REGION Network 73: SN51_N0063
   RUNG wire#powerrail
      Contact( "AlwaysTRUE" )
      Contact( "ZAUX".SN51_N0063 )
      Coil( "00_Commissioning"."n0063-lv006-el001-k30001_SN51" )
   END_RUNG
   // the same network as SCL:
   "00_Commissioning"."n0063-lv006-el001-k30001_SN51" := "AlwaysTRUE" AND "ZAUX".SN51_N0063;
END_REGION

REGION Network 74: SN51_N0066
   RUNG wire#powerrail
      Contact( "AlwaysTRUE" )
      Contact( "ZAUX".SN51_N0066 )
      Coil( "00_Commissioning"."n0066-uc21-el001-k30001_SN51" )
   END_RUNG
   // the same network as SCL:
   "00_Commissioning"."n0066-uc21-el001-k30001_SN51" := "AlwaysTRUE" AND "ZAUX".SN51_N0066;
END_REGION

REGION Network 75: SN51_N0067
   RUNG wire#powerrail
      Contact( "AlwaysTRUE" )
      Contact( "ZAUX".SN51_N0067 )
      Coil( "00_Commissioning"."n0067-uc214-xn10_SN51" )
   END_RUNG
   // the same network as SCL:
   "00_Commissioning"."n0067-uc214-xn10_SN51" := "AlwaysTRUE" AND "ZAUX".SN51_N0067;
END_REGION

REGION Network 76: SN51_N0070
   RUNG wire#powerrail
      Contact( "AlwaysTRUE" )
      Contact( "ZAUX".SN51_N0070 )
      Coil( "00_Commissioning"."n0070-uf31-el001-k30001_SN51" )
   END_RUNG
   // the same network as SCL:
   "00_Commissioning"."n0070-uf31-el001-k30001_SN51" := "AlwaysTRUE" AND "ZAUX".SN51_N0070;
END_REGION

REGION Network 77: SN51_N0071
   RUNG wire#powerrail
      Contact( "AlwaysTRUE" )
      Contact( "ZAUX".SN51_N0071 )
      Coil( "00_Commissioning"."n0070-uf31-el001-k30001_SN51" )
   END_RUNG
   // the same network as SCL:
   "00_Commissioning"."n0070-uf31-el001-k30001_SN51" := "AlwaysTRUE" AND "ZAUX".SN51_N0071;
END_REGION

REGION Network 78: SN51_N0072
   RUNG wire#powerrail
      Contact( "AlwaysTRUE" )
      Contact( "ZAUX".SN51_N0072 )
      Coil( "00_Commissioning"."n0072-uf51-el001-k30001_SN51" )
   END_RUNG
   // the same network as SCL:
   "00_Commissioning"."n0072-uf51-el001-k30001_SN51" := "AlwaysTRUE" AND "ZAUX".SN51_N0072;
END_REGION

REGION Network 79: SN51_N0080
   RUNG wire#powerrail
      Contact( "AlwaysTRUE" )
      Contact( "ZAUX".SN51_N0080 )
      Coil( "00_Commissioning"."n0080-uf511-xn10_SN51" )
   END_RUNG
   // the same network as SCL:
   "00_Commissioning"."n0080-uf511-xn10_SN51" := "AlwaysTRUE" AND "ZAUX".SN51_N0080;
END_REGION

REGION Network 80: SN51_N0073
   RUNG wire#powerrail
      Contact( "AlwaysTRUE" )
      Contact( "ZAUX".SN51_N0073 )
      Coil( "00_Commissioning"."n0073-ifg31-el001-k30001_SN51" )
   END_RUNG
   // the same network as SCL:
   "00_Commissioning"."n0073-ifg31-el001-k30001_SN51" := "AlwaysTRUE" AND "ZAUX".SN51_N0073;
END_REGION

REGION Network 81: SN51_N0074
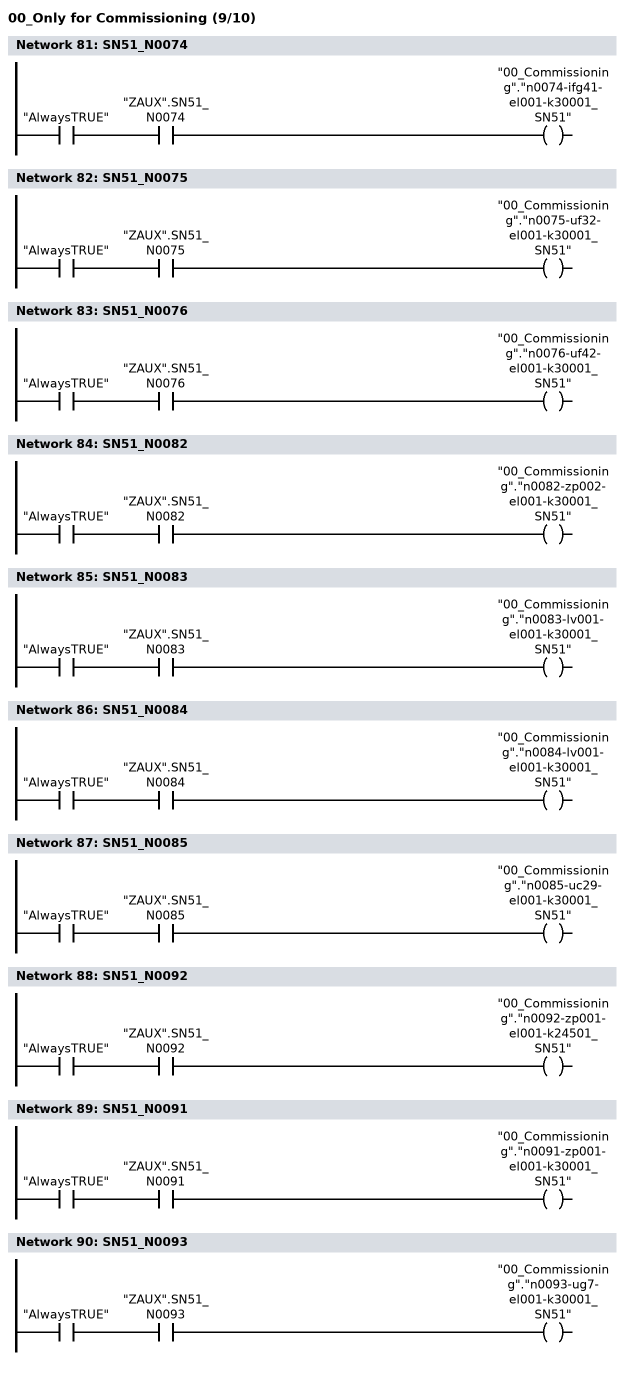
   RUNG wire#powerrail
      Contact( "AlwaysTRUE" )
      Contact( "ZAUX".SN51_N0074 )
      Coil( "00_Commissioning"."n0074-ifg41-el001-k30001_SN51" )
   END_RUNG
   // the same network as SCL:
   "00_Commissioning"."n0074-ifg41-el001-k30001_SN51" := "AlwaysTRUE" AND "ZAUX".SN51_N0074;
END_REGION

REGION Network 82: SN51_N0075
   RUNG wire#powerrail
      Contact( "AlwaysTRUE" )
      Contact( "ZAUX".SN51_N0075 )
      Coil( "00_Commissioning"."n0075-uf32-el001-k30001_SN51" )
   END_RUNG
   // the same network as SCL:
   "00_Commissioning"."n0075-uf32-el001-k30001_SN51" := "AlwaysTRUE" AND "ZAUX".SN51_N0075;
END_REGION

REGION Network 83: SN51_N0076
   RUNG wire#powerrail
      Contact( "AlwaysTRUE" )
      Contact( "ZAUX".SN51_N0076 )
      Coil( "00_Commissioning"."n0076-uf42-el001-k30001_SN51" )
   END_RUNG
   // the same network as SCL:
   "00_Commissioning"."n0076-uf42-el001-k30001_SN51" := "AlwaysTRUE" AND "ZAUX".SN51_N0076;
END_REGION

REGION Network 84: SN51_N0082
   RUNG wire#powerrail
      Contact( "AlwaysTRUE" )
      Contact( "ZAUX".SN51_N0082 )
      Coil( "00_Commissioning"."n0082-zp002-el001-k30001_SN51" )
   END_RUNG
   // the same network as SCL:
   "00_Commissioning"."n0082-zp002-el001-k30001_SN51" := "AlwaysTRUE" AND "ZAUX".SN51_N0082;
END_REGION

REGION Network 85: SN51_N0083
   RUNG wire#powerrail
      Contact( "AlwaysTRUE" )
      Contact( "ZAUX".SN51_N0083 )
      Coil( "00_Commissioning"."n0083-lv001-el001-k30001_SN51" )
   END_RUNG
   // the same network as SCL:
   "00_Commissioning"."n0083-lv001-el001-k30001_SN51" := "AlwaysTRUE" AND "ZAUX".SN51_N0083;
END_REGION

REGION Network 86: SN51_N0084
   RUNG wire#powerrail
      Contact( "AlwaysTRUE" )
      Contact( "ZAUX".SN51_N0084 )
      Coil( "00_Commissioning"."n0084-lv001-el001-k30001_SN51" )
   END_RUNG
   // the same network as SCL:
   "00_Commissioning"."n0084-lv001-el001-k30001_SN51" := "AlwaysTRUE" AND "ZAUX".SN51_N0084;
END_REGION

REGION Network 87: SN51_N0085
   RUNG wire#powerrail
      Contact( "AlwaysTRUE" )
      Contact( "ZAUX".SN51_N0085 )
      Coil( "00_Commissioning"."n0085-uc29-el001-k30001_SN51" )
   END_RUNG
   // the same network as SCL:
   "00_Commissioning"."n0085-uc29-el001-k30001_SN51" := "AlwaysTRUE" AND "ZAUX".SN51_N0085;
END_REGION

REGION Network 88: SN51_N0092
   RUNG wire#powerrail
      Contact( "AlwaysTRUE" )
      Contact( "ZAUX".SN51_N0092 )
      Coil( "00_Commissioning"."n0092-zp001-el001-k24501_SN51" )
   END_RUNG
   // the same network as SCL:
   "00_Commissioning"."n0092-zp001-el001-k24501_SN51" := "AlwaysTRUE" AND "ZAUX".SN51_N0092;
END_REGION

REGION Network 89: SN51_N0091
   RUNG wire#powerrail
      Contact( "AlwaysTRUE" )
      Contact( "ZAUX".SN51_N0091 )
      Coil( "00_Commissioning"."n0091-zp001-el001-k30001_SN51" )
   END_RUNG
   // the same network as SCL:
   "00_Commissioning"."n0091-zp001-el001-k30001_SN51" := "AlwaysTRUE" AND "ZAUX".SN51_N0091;
END_REGION

REGION Network 90: SN51_N0093
   RUNG wire#powerrail
      Contact( "AlwaysTRUE" )
      Contact( "ZAUX".SN51_N0093 )
      Coil( "00_Commissioning"."n0093-ug7-el001-k30001_SN51" )
   END_RUNG
   // the same network as SCL:
   "00_Commissioning"."n0093-ug7-el001-k30001_SN51" := "AlwaysTRUE" AND "ZAUX".SN51_N0093;
END_REGION

REGION Network 91: SN51_N0094
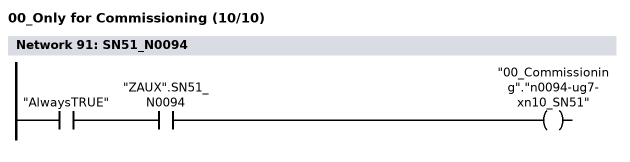
   RUNG wire#powerrail
      Contact( "AlwaysTRUE" )
      Contact( "ZAUX".SN51_N0094 )
      Coil( "00_Commissioning"."n0094-ug7-xn10_SN51" )
   END_RUNG
   // the same network as SCL:
   "00_Commissioning"."n0094-ug7-xn10_SN51" := "AlwaysTRUE" AND "ZAUX".SN51_N0094;
END_REGION
END_FUNCTION

FUNCTION "01_Settings" : Void   // FC2, F_FBD
{ S7_Optimized_Access := 'TRUE' }
VERSION : 0.1
BEGIN

REGION Network 1: To be used in case of overall settings
   // for example in case of Tristate diagnostic
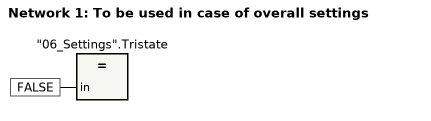
   "06_Settings".Tristate := FALSE;
END_REGION
END_FUNCTION

FUNCTION "02_EM Push Button" : Void   // FC3, F_LAD
TITLE = Mirror PB
{ S7_Optimized_Access := 'TRUE' }
VERSION : 0.1
BEGIN

REGION Network 1: 50.005 | n0005-zp001-el001-k40001_SN50 [1]
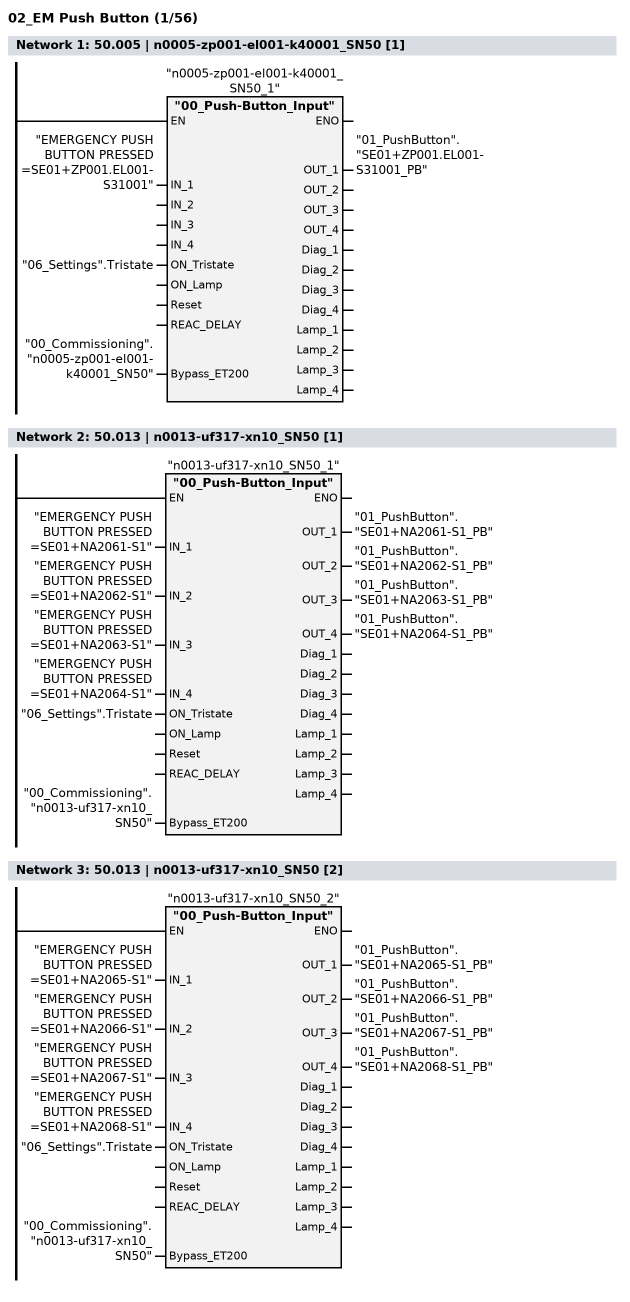
   RUNG wire#powerrail
      "n0005-zp001-el001-k40001_SN50_1"(IN_1 := "EMERGENCY PUSH BUTTON PRESSED =SE01+ZP001.EL001-S31001", IN_2 :=, IN_3 :=, IN_4 :=, ON_Tristate := "06_Settings".Tristate, ON_Lamp :=, Reset :=, REAC_DELAY :=, Bypass_ET200 := "00_Commissioning"."n0005-zp001-el001-k40001_SN50", OUT_1 => "01_PushButton"."SE01+ZP001.EL001-S31001_PB", OUT_2 =>, OUT_3 =>, OUT_4 =>, Diag_1 =>, Diag_2 =>, Diag_3 =>, Diag_4 =>, Lamp_1 =>, Lamp_2 =>, Lamp_3 =>, Lamp_4 =>)
   END_RUNG
   // the same network as SCL:
   "n0005-zp001-el001-k40001_SN50_1"(IN_1 := "EMERGENCY PUSH BUTTON PRESSED =SE01+ZP001.EL001-S31001",   // "00_Push-Button_Input"
                           ON_Tristate := "06_Settings".Tristate,
                           Bypass_ET200 := "00_Commissioning"."n0005-zp001-el001-k40001_SN50",
                           OUT_1 => "01_PushButton"."SE01+ZP001.EL001-S31001_PB");
END_REGION

REGION Network 2: 50.013 | n0013-uf317-xn10_SN50 [1]
   RUNG wire#powerrail
      "n0013-uf317-xn10_SN50_1"(IN_1 := "EMERGENCY PUSH BUTTON PRESSED =SE01+NA2061-S1", IN_2 := "EMERGENCY PUSH BUTTON PRESSED =SE01+NA2062-S1", IN_3 := "EMERGENCY PUSH BUTTON PRESSED =SE01+NA2063-S1", IN_4 := "EMERGENCY PUSH BUTTON PRESSED =SE01+NA2064-S1", ON_Tristate := "06_Settings".Tristate, ON_Lamp :=, Reset :=, REAC_DELAY :=, Bypass_ET200 := "00_Commissioning"."n0013-uf317-xn10_SN50", OUT_1 => "01_PushButton"."SE01+NA2061-S1_PB", OUT_2 => "01_PushButton"."SE01+NA2062-S1_PB", OUT_3 => "01_PushButton"."SE01+NA2063-S1_PB", OUT_4 => "01_PushButton"."SE01+NA2064-S1_PB", Diag_1 =>, Diag_2 =>, Diag_3 =>, Diag_4 =>, Lamp_1 =>, Lamp_2 =>, Lamp_3 =>, Lamp_4 =>)
   END_RUNG
   // the same network as SCL:
   "n0013-uf317-xn10_SN50_1"(IN_1 := "EMERGENCY PUSH BUTTON PRESSED =SE01+NA2061-S1",   // "00_Push-Button_Input"
                           IN_2 := "EMERGENCY PUSH BUTTON PRESSED =SE01+NA2062-S1",
                           IN_3 := "EMERGENCY PUSH BUTTON PRESSED =SE01+NA2063-S1",
                           IN_4 := "EMERGENCY PUSH BUTTON PRESSED =SE01+NA2064-S1",
                           ON_Tristate := "06_Settings".Tristate,
                           Bypass_ET200 := "00_Commissioning"."n0013-uf317-xn10_SN50",
                           OUT_1 => "01_PushButton"."SE01+NA2061-S1_PB",
                           OUT_2 => "01_PushButton"."SE01+NA2062-S1_PB",
                           OUT_3 => "01_PushButton"."SE01+NA2063-S1_PB",
                           OUT_4 => "01_PushButton"."SE01+NA2064-S1_PB");
END_REGION

REGION Network 3: 50.013 | n0013-uf317-xn10_SN50 [2]
   RUNG wire#powerrail
      "n0013-uf317-xn10_SN50_2"(IN_1 := "EMERGENCY PUSH BUTTON PRESSED =SE01+NA2065-S1", IN_2 := "EMERGENCY PUSH BUTTON PRESSED =SE01+NA2066-S1", IN_3 := "EMERGENCY PUSH BUTTON PRESSED =SE01+NA2067-S1", IN_4 := "EMERGENCY PUSH BUTTON PRESSED =SE01+NA2068-S1", ON_Tristate := "06_Settings".Tristate, ON_Lamp :=, Reset :=, REAC_DELAY :=, Bypass_ET200 := "00_Commissioning"."n0013-uf317-xn10_SN50", OUT_1 => "01_PushButton"."SE01+NA2065-S1_PB", OUT_2 => "01_PushButton"."SE01+NA2066-S1_PB", OUT_3 => "01_PushButton"."SE01+NA2067-S1_PB", OUT_4 => "01_PushButton"."SE01+NA2068-S1_PB", Diag_1 =>, Diag_2 =>, Diag_3 =>, Diag_4 =>, Lamp_1 =>, Lamp_2 =>, Lamp_3 =>, Lamp_4 =>)
   END_RUNG
   // the same network as SCL:
   "n0013-uf317-xn10_SN50_2"(IN_1 := "EMERGENCY PUSH BUTTON PRESSED =SE01+NA2065-S1",   // "00_Push-Button_Input"
                           IN_2 := "EMERGENCY PUSH BUTTON PRESSED =SE01+NA2066-S1",
                           IN_3 := "EMERGENCY PUSH BUTTON PRESSED =SE01+NA2067-S1",
                           IN_4 := "EMERGENCY PUSH BUTTON PRESSED =SE01+NA2068-S1",
                           ON_Tristate := "06_Settings".Tristate,
                           Bypass_ET200 := "00_Commissioning"."n0013-uf317-xn10_SN50",
                           OUT_1 => "01_PushButton"."SE01+NA2065-S1_PB",
                           OUT_2 => "01_PushButton"."SE01+NA2066-S1_PB",
                           OUT_3 => "01_PushButton"."SE01+NA2067-S1_PB",
                           OUT_4 => "01_PushButton"."SE01+NA2068-S1_PB");
END_REGION

REGION Network 4: 50.015 | n0015-uc16-el001-k30001_SN50 [1]
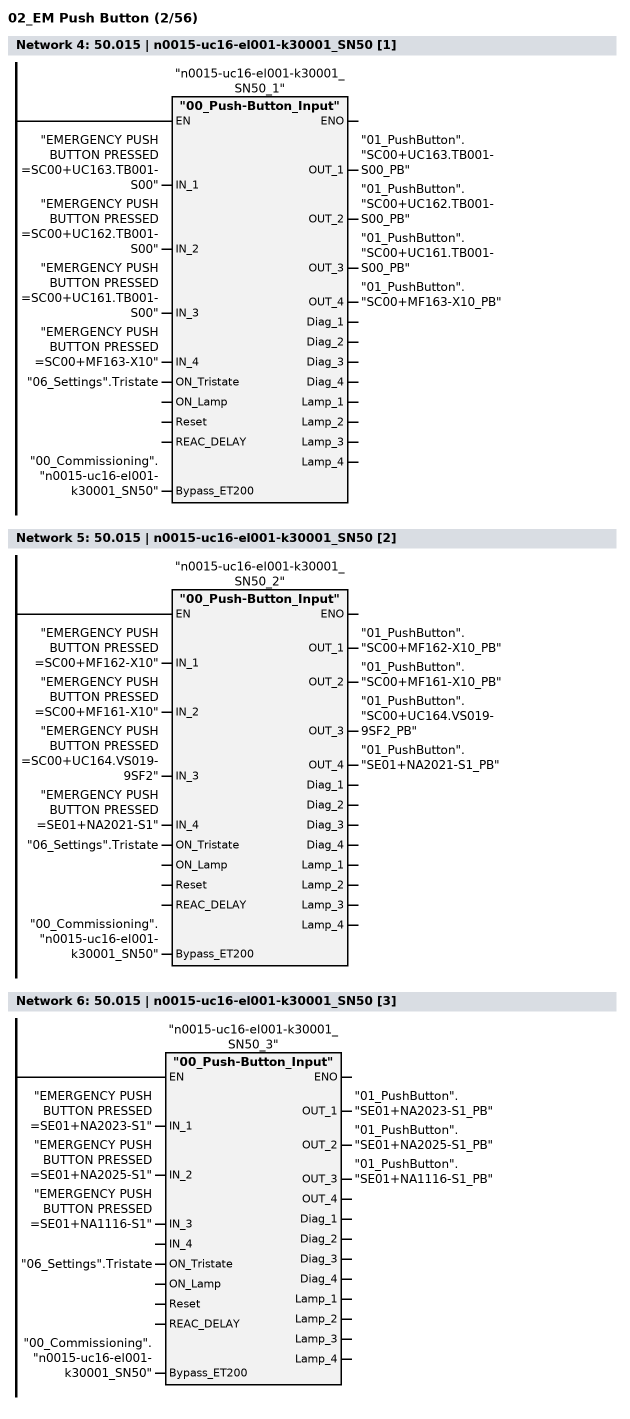
   RUNG wire#powerrail
      "n0015-uc16-el001-k30001_SN50_1"(IN_1 := "EMERGENCY PUSH BUTTON PRESSED =SC00+UC163.TB001-S00", IN_2 := "EMERGENCY PUSH BUTTON PRESSED =SC00+UC162.TB001-S00", IN_3 := "EMERGENCY PUSH BUTTON PRESSED =SC00+UC161.TB001-S00", IN_4 := "EMERGENCY PUSH BUTTON PRESSED =SC00+MF163-X10", ON_Tristate := "06_Settings".Tristate, ON_Lamp :=, Reset :=, REAC_DELAY :=, Bypass_ET200 := "00_Commissioning"."n0015-uc16-el001-k30001_SN50", OUT_1 => "01_PushButton"."SC00+UC163.TB001-S00_PB", OUT_2 => "01_PushButton"."SC00+UC162.TB001-S00_PB", OUT_3 => "01_PushButton"."SC00+UC161.TB001-S00_PB", OUT_4 => "01_PushButton"."SC00+MF163-X10_PB", Diag_1 =>, Diag_2 =>, Diag_3 =>, Diag_4 =>, Lamp_1 =>, Lamp_2 =>, Lamp_3 =>, Lamp_4 =>)
   END_RUNG
   // the same network as SCL:
   "n0015-uc16-el001-k30001_SN50_1"(IN_1 := "EMERGENCY PUSH BUTTON PRESSED =SC00+UC163.TB001-S00",   // "00_Push-Button_Input"
                           IN_2 := "EMERGENCY PUSH BUTTON PRESSED =SC00+UC162.TB001-S00",
                           IN_3 := "EMERGENCY PUSH BUTTON PRESSED =SC00+UC161.TB001-S00",
                           IN_4 := "EMERGENCY PUSH BUTTON PRESSED =SC00+MF163-X10",
                           ON_Tristate := "06_Settings".Tristate,
                           Bypass_ET200 := "00_Commissioning"."n0015-uc16-el001-k30001_SN50",
                           OUT_1 => "01_PushButton"."SC00+UC163.TB001-S00_PB",
                           OUT_2 => "01_PushButton"."SC00+UC162.TB001-S00_PB",
                           OUT_3 => "01_PushButton"."SC00+UC161.TB001-S00_PB",
                           OUT_4 => "01_PushButton"."SC00+MF163-X10_PB");
END_REGION

REGION Network 5: 50.015 | n0015-uc16-el001-k30001_SN50 [2]
   RUNG wire#powerrail
      "n0015-uc16-el001-k30001_SN50_2"(IN_1 := "EMERGENCY PUSH BUTTON PRESSED =SC00+MF162-X10", IN_2 := "EMERGENCY PUSH BUTTON PRESSED =SC00+MF161-X10", IN_3 := "EMERGENCY PUSH BUTTON PRESSED =SC00+UC164.VS019-9SF2", IN_4 := "EMERGENCY PUSH BUTTON PRESSED =SE01+NA2021-S1", ON_Tristate := "06_Settings".Tristate, ON_Lamp :=, Reset :=, REAC_DELAY :=, Bypass_ET200 := "00_Commissioning"."n0015-uc16-el001-k30001_SN50", OUT_1 => "01_PushButton"."SC00+MF162-X10_PB", OUT_2 => "01_PushButton"."SC00+MF161-X10_PB", OUT_3 => "01_PushButton"."SC00+UC164.VS019-9SF2_PB", OUT_4 => "01_PushButton"."SE01+NA2021-S1_PB", Diag_1 =>, Diag_2 =>, Diag_3 =>, Diag_4 =>, Lamp_1 =>, Lamp_2 =>, Lamp_3 =>, Lamp_4 =>)
   END_RUNG
   // the same network as SCL:
   "n0015-uc16-el001-k30001_SN50_2"(IN_1 := "EMERGENCY PUSH BUTTON PRESSED =SC00+MF162-X10",   // "00_Push-Button_Input"
                           IN_2 := "EMERGENCY PUSH BUTTON PRESSED =SC00+MF161-X10",
                           IN_3 := "EMERGENCY PUSH BUTTON PRESSED =SC00+UC164.VS019-9SF2",
                           IN_4 := "EMERGENCY PUSH BUTTON PRESSED =SE01+NA2021-S1",
                           ON_Tristate := "06_Settings".Tristate,
                           Bypass_ET200 := "00_Commissioning"."n0015-uc16-el001-k30001_SN50",
                           OUT_1 => "01_PushButton"."SC00+MF162-X10_PB",
                           OUT_2 => "01_PushButton"."SC00+MF161-X10_PB",
                           OUT_3 => "01_PushButton"."SC00+UC164.VS019-9SF2_PB",
                           OUT_4 => "01_PushButton"."SE01+NA2021-S1_PB");
END_REGION

REGION Network 6: 50.015 | n0015-uc16-el001-k30001_SN50 [3]
   RUNG wire#powerrail
      "n0015-uc16-el001-k30001_SN50_3"(IN_1 := "EMERGENCY PUSH BUTTON PRESSED =SE01+NA2023-S1", IN_2 := "EMERGENCY PUSH BUTTON PRESSED =SE01+NA2025-S1", IN_3 := "EMERGENCY PUSH BUTTON PRESSED =SE01+NA1116-S1", IN_4 :=, ON_Tristate := "06_Settings".Tristate, ON_Lamp :=, Reset :=, REAC_DELAY :=, Bypass_ET200 := "00_Commissioning"."n0015-uc16-el001-k30001_SN50", OUT_1 => "01_PushButton"."SE01+NA2023-S1_PB", OUT_2 => "01_PushButton"."SE01+NA2025-S1_PB", OUT_3 => "01_PushButton"."SE01+NA1116-S1_PB", OUT_4 =>, Diag_1 =>, Diag_2 =>, Diag_3 =>, Diag_4 =>, Lamp_1 =>, Lamp_2 =>, Lamp_3 =>, Lamp_4 =>)
   END_RUNG
   // the same network as SCL:
   "n0015-uc16-el001-k30001_SN50_3"(IN_1 := "EMERGENCY PUSH BUTTON PRESSED =SE01+NA2023-S1",   // "00_Push-Button_Input"
                           IN_2 := "EMERGENCY PUSH BUTTON PRESSED =SE01+NA2025-S1",
                           IN_3 := "EMERGENCY PUSH BUTTON PRESSED =SE01+NA1116-S1",
                           ON_Tristate := "06_Settings".Tristate,
                           Bypass_ET200 := "00_Commissioning"."n0015-uc16-el001-k30001_SN50",
                           OUT_1 => "01_PushButton"."SE01+NA2023-S1_PB",
                           OUT_2 => "01_PushButton"."SE01+NA2025-S1_PB",
                           OUT_3 => "01_PushButton"."SE01+NA1116-S1_PB");
END_REGION

REGION Network 7: 50.016 | n0016-uc164-xn10_SN50 [1]
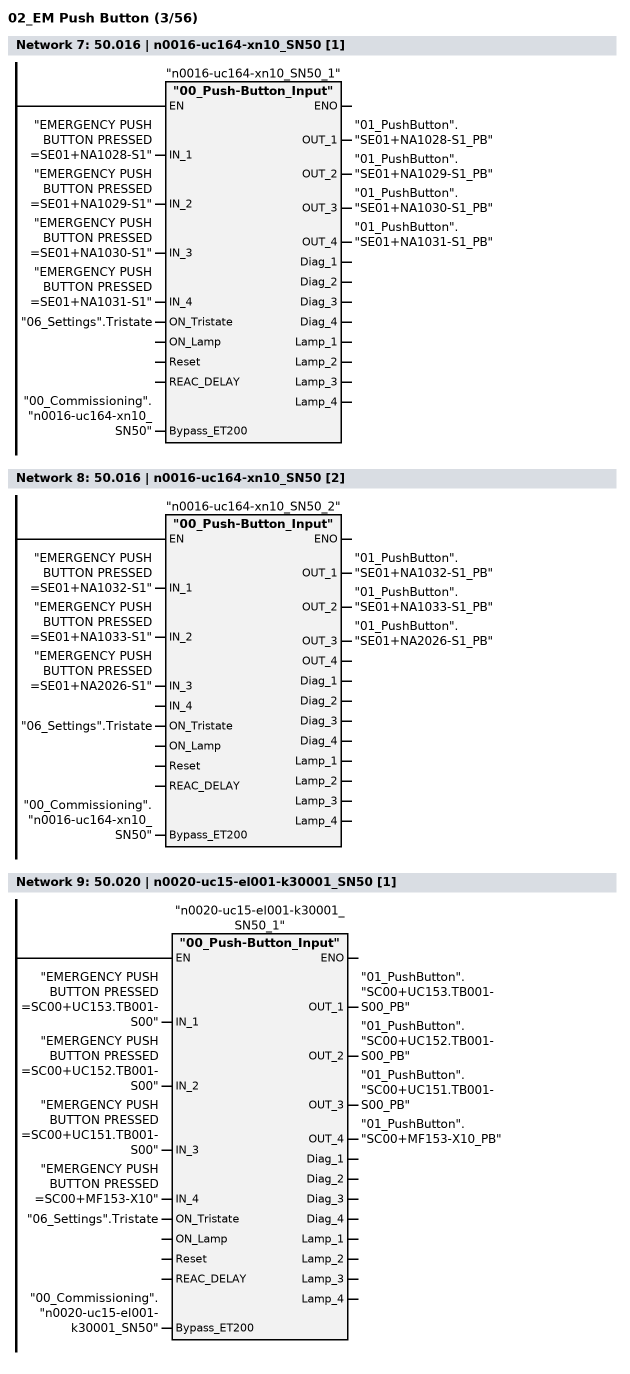
   RUNG wire#powerrail
      "n0016-uc164-xn10_SN50_1"(IN_1 := "EMERGENCY PUSH BUTTON PRESSED =SE01+NA1028-S1", IN_2 := "EMERGENCY PUSH BUTTON PRESSED =SE01+NA1029-S1", IN_3 := "EMERGENCY PUSH BUTTON PRESSED =SE01+NA1030-S1", IN_4 := "EMERGENCY PUSH BUTTON PRESSED =SE01+NA1031-S1", ON_Tristate := "06_Settings".Tristate, ON_Lamp :=, Reset :=, REAC_DELAY :=, Bypass_ET200 := "00_Commissioning"."n0016-uc164-xn10_SN50", OUT_1 => "01_PushButton"."SE01+NA1028-S1_PB", OUT_2 => "01_PushButton"."SE01+NA1029-S1_PB", OUT_3 => "01_PushButton"."SE01+NA1030-S1_PB", OUT_4 => "01_PushButton"."SE01+NA1031-S1_PB", Diag_1 =>, Diag_2 =>, Diag_3 =>, Diag_4 =>, Lamp_1 =>, Lamp_2 =>, Lamp_3 =>, Lamp_4 =>)
   END_RUNG
   // the same network as SCL:
   "n0016-uc164-xn10_SN50_1"(IN_1 := "EMERGENCY PUSH BUTTON PRESSED =SE01+NA1028-S1",   // "00_Push-Button_Input"
                           IN_2 := "EMERGENCY PUSH BUTTON PRESSED =SE01+NA1029-S1",
                           IN_3 := "EMERGENCY PUSH BUTTON PRESSED =SE01+NA1030-S1",
                           IN_4 := "EMERGENCY PUSH BUTTON PRESSED =SE01+NA1031-S1",
                           ON_Tristate := "06_Settings".Tristate,
                           Bypass_ET200 := "00_Commissioning"."n0016-uc164-xn10_SN50",
                           OUT_1 => "01_PushButton"."SE01+NA1028-S1_PB",
                           OUT_2 => "01_PushButton"."SE01+NA1029-S1_PB",
                           OUT_3 => "01_PushButton"."SE01+NA1030-S1_PB",
                           OUT_4 => "01_PushButton"."SE01+NA1031-S1_PB");
END_REGION

REGION Network 8: 50.016 | n0016-uc164-xn10_SN50 [2]
   RUNG wire#powerrail
      "n0016-uc164-xn10_SN50_2"(IN_1 := "EMERGENCY PUSH BUTTON PRESSED =SE01+NA1032-S1", IN_2 := "EMERGENCY PUSH BUTTON PRESSED =SE01+NA1033-S1", IN_3 := "EMERGENCY PUSH BUTTON PRESSED =SE01+NA2026-S1", IN_4 :=, ON_Tristate := "06_Settings".Tristate, ON_Lamp :=, Reset :=, REAC_DELAY :=, Bypass_ET200 := "00_Commissioning"."n0016-uc164-xn10_SN50", OUT_1 => "01_PushButton"."SE01+NA1032-S1_PB", OUT_2 => "01_PushButton"."SE01+NA1033-S1_PB", OUT_3 => "01_PushButton"."SE01+NA2026-S1_PB", OUT_4 =>, Diag_1 =>, Diag_2 =>, Diag_3 =>, Diag_4 =>, Lamp_1 =>, Lamp_2 =>, Lamp_3 =>, Lamp_4 =>)
   END_RUNG
   // the same network as SCL:
   "n0016-uc164-xn10_SN50_2"(IN_1 := "EMERGENCY PUSH BUTTON PRESSED =SE01+NA1032-S1",   // "00_Push-Button_Input"
                           IN_2 := "EMERGENCY PUSH BUTTON PRESSED =SE01+NA1033-S1",
                           IN_3 := "EMERGENCY PUSH BUTTON PRESSED =SE01+NA2026-S1",
                           ON_Tristate := "06_Settings".Tristate,
                           Bypass_ET200 := "00_Commissioning"."n0016-uc164-xn10_SN50",
                           OUT_1 => "01_PushButton"."SE01+NA1032-S1_PB",
                           OUT_2 => "01_PushButton"."SE01+NA1033-S1_PB",
                           OUT_3 => "01_PushButton"."SE01+NA2026-S1_PB");
END_REGION

REGION Network 9: 50.020 | n0020-uc15-el001-k30001_SN50 [1]
   RUNG wire#powerrail
      "n0020-uc15-el001-k30001_SN50_1"(IN_1 := "EMERGENCY PUSH BUTTON PRESSED =SC00+UC153.TB001-S00", IN_2 := "EMERGENCY PUSH BUTTON PRESSED =SC00+UC152.TB001-S00", IN_3 := "EMERGENCY PUSH BUTTON PRESSED =SC00+UC151.TB001-S00", IN_4 := "EMERGENCY PUSH BUTTON PRESSED =SC00+MF153-X10", ON_Tristate := "06_Settings".Tristate, ON_Lamp :=, Reset :=, REAC_DELAY :=, Bypass_ET200 := "00_Commissioning"."n0020-uc15-el001-k30001_SN50", OUT_1 => "01_PushButton"."SC00+UC153.TB001-S00_PB", OUT_2 => "01_PushButton"."SC00+UC152.TB001-S00_PB", OUT_3 => "01_PushButton"."SC00+UC151.TB001-S00_PB", OUT_4 => "01_PushButton"."SC00+MF153-X10_PB", Diag_1 =>, Diag_2 =>, Diag_3 =>, Diag_4 =>, Lamp_1 =>, Lamp_2 =>, Lamp_3 =>, Lamp_4 =>)
   END_RUNG
   // the same network as SCL:
   "n0020-uc15-el001-k30001_SN50_1"(IN_1 := "EMERGENCY PUSH BUTTON PRESSED =SC00+UC153.TB001-S00",   // "00_Push-Button_Input"
                           IN_2 := "EMERGENCY PUSH BUTTON PRESSED =SC00+UC152.TB001-S00",
                           IN_3 := "EMERGENCY PUSH BUTTON PRESSED =SC00+UC151.TB001-S00",
                           IN_4 := "EMERGENCY PUSH BUTTON PRESSED =SC00+MF153-X10",
                           ON_Tristate := "06_Settings".Tristate,
                           Bypass_ET200 := "00_Commissioning"."n0020-uc15-el001-k30001_SN50",
                           OUT_1 => "01_PushButton"."SC00+UC153.TB001-S00_PB",
                           OUT_2 => "01_PushButton"."SC00+UC152.TB001-S00_PB",
                           OUT_3 => "01_PushButton"."SC00+UC151.TB001-S00_PB",
                           OUT_4 => "01_PushButton"."SC00+MF153-X10_PB");
END_REGION

REGION Network 10: 50.020 | n0020-uc15-el001-k30001_SN50 [2]
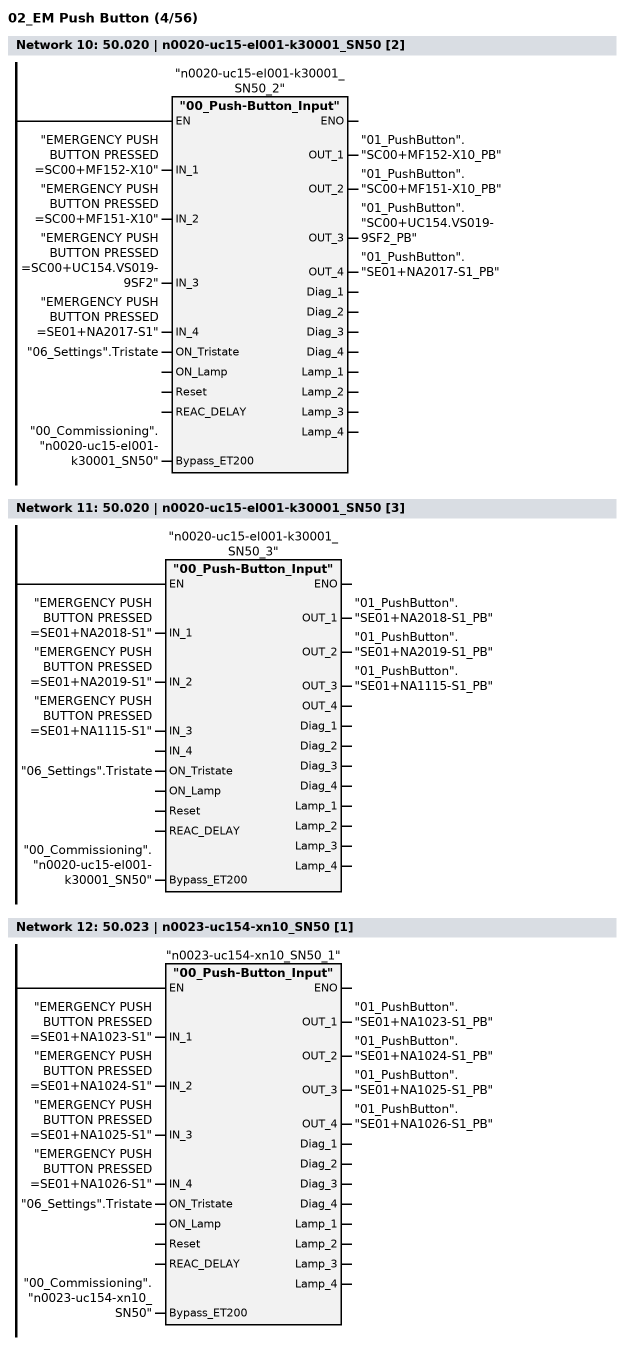
   RUNG wire#powerrail
      "n0020-uc15-el001-k30001_SN50_2"(IN_1 := "EMERGENCY PUSH BUTTON PRESSED =SC00+MF152-X10", IN_2 := "EMERGENCY PUSH BUTTON PRESSED =SC00+MF151-X10", IN_3 := "EMERGENCY PUSH BUTTON PRESSED =SC00+UC154.VS019-9SF2", IN_4 := "EMERGENCY PUSH BUTTON PRESSED =SE01+NA2017-S1", ON_Tristate := "06_Settings".Tristate, ON_Lamp :=, Reset :=, REAC_DELAY :=, Bypass_ET200 := "00_Commissioning"."n0020-uc15-el001-k30001_SN50", OUT_1 => "01_PushButton"."SC00+MF152-X10_PB", OUT_2 => "01_PushButton"."SC00+MF151-X10_PB", OUT_3 => "01_PushButton"."SC00+UC154.VS019-9SF2_PB", OUT_4 => "01_PushButton"."SE01+NA2017-S1_PB", Diag_1 =>, Diag_2 =>, Diag_3 =>, Diag_4 =>, Lamp_1 =>, Lamp_2 =>, Lamp_3 =>, Lamp_4 =>)
   END_RUNG
   // the same network as SCL:
   "n0020-uc15-el001-k30001_SN50_2"(IN_1 := "EMERGENCY PUSH BUTTON PRESSED =SC00+MF152-X10",   // "00_Push-Button_Input"
                           IN_2 := "EMERGENCY PUSH BUTTON PRESSED =SC00+MF151-X10",
                           IN_3 := "EMERGENCY PUSH BUTTON PRESSED =SC00+UC154.VS019-9SF2",
                           IN_4 := "EMERGENCY PUSH BUTTON PRESSED =SE01+NA2017-S1",
                           ON_Tristate := "06_Settings".Tristate,
                           Bypass_ET200 := "00_Commissioning"."n0020-uc15-el001-k30001_SN50",
                           OUT_1 => "01_PushButton"."SC00+MF152-X10_PB",
                           OUT_2 => "01_PushButton"."SC00+MF151-X10_PB",
                           OUT_3 => "01_PushButton"."SC00+UC154.VS019-9SF2_PB",
                           OUT_4 => "01_PushButton"."SE01+NA2017-S1_PB");
END_REGION

REGION Network 11: 50.020 | n0020-uc15-el001-k30001_SN50 [3]
   RUNG wire#powerrail
      "n0020-uc15-el001-k30001_SN50_3"(IN_1 := "EMERGENCY PUSH BUTTON PRESSED =SE01+NA2018-S1", IN_2 := "EMERGENCY PUSH BUTTON PRESSED =SE01+NA2019-S1", IN_3 := "EMERGENCY PUSH BUTTON PRESSED =SE01+NA1115-S1", IN_4 :=, ON_Tristate := "06_Settings".Tristate, ON_Lamp :=, Reset :=, REAC_DELAY :=, Bypass_ET200 := "00_Commissioning"."n0020-uc15-el001-k30001_SN50", OUT_1 => "01_PushButton"."SE01+NA2018-S1_PB", OUT_2 => "01_PushButton"."SE01+NA2019-S1_PB", OUT_3 => "01_PushButton"."SE01+NA1115-S1_PB", OUT_4 =>, Diag_1 =>, Diag_2 =>, Diag_3 =>, Diag_4 =>, Lamp_1 =>, Lamp_2 =>, Lamp_3 =>, Lamp_4 =>)
   END_RUNG
   // the same network as SCL:
   "n0020-uc15-el001-k30001_SN50_3"(IN_1 := "EMERGENCY PUSH BUTTON PRESSED =SE01+NA2018-S1",   // "00_Push-Button_Input"
                           IN_2 := "EMERGENCY PUSH BUTTON PRESSED =SE01+NA2019-S1",
                           IN_3 := "EMERGENCY PUSH BUTTON PRESSED =SE01+NA1115-S1",
                           ON_Tristate := "06_Settings".Tristate,
                           Bypass_ET200 := "00_Commissioning"."n0020-uc15-el001-k30001_SN50",
                           OUT_1 => "01_PushButton"."SE01+NA2018-S1_PB",
                           OUT_2 => "01_PushButton"."SE01+NA2019-S1_PB",
                           OUT_3 => "01_PushButton"."SE01+NA1115-S1_PB");
END_REGION

REGION Network 12: 50.023 | n0023-uc154-xn10_SN50 [1]
   RUNG wire#powerrail
      "n0023-uc154-xn10_SN50_1"(IN_1 := "EMERGENCY PUSH BUTTON PRESSED =SE01+NA1023-S1", IN_2 := "EMERGENCY PUSH BUTTON PRESSED =SE01+NA1024-S1", IN_3 := "EMERGENCY PUSH BUTTON PRESSED =SE01+NA1025-S1", IN_4 := "EMERGENCY PUSH BUTTON PRESSED =SE01+NA1026-S1", ON_Tristate := "06_Settings".Tristate, ON_Lamp :=, Reset :=, REAC_DELAY :=, Bypass_ET200 := "00_Commissioning"."n0023-uc154-xn10_SN50", OUT_1 => "01_PushButton"."SE01+NA1023-S1_PB", OUT_2 => "01_PushButton"."SE01+NA1024-S1_PB", OUT_3 => "01_PushButton"."SE01+NA1025-S1_PB", OUT_4 => "01_PushButton"."SE01+NA1026-S1_PB", Diag_1 =>, Diag_2 =>, Diag_3 =>, Diag_4 =>, Lamp_1 =>, Lamp_2 =>, Lamp_3 =>, Lamp_4 =>)
   END_RUNG
   // the same network as SCL:
   "n0023-uc154-xn10_SN50_1"(IN_1 := "EMERGENCY PUSH BUTTON PRESSED =SE01+NA1023-S1",   // "00_Push-Button_Input"
                           IN_2 := "EMERGENCY PUSH BUTTON PRESSED =SE01+NA1024-S1",
                           IN_3 := "EMERGENCY PUSH BUTTON PRESSED =SE01+NA1025-S1",
                           IN_4 := "EMERGENCY PUSH BUTTON PRESSED =SE01+NA1026-S1",
                           ON_Tristate := "06_Settings".Tristate,
                           Bypass_ET200 := "00_Commissioning"."n0023-uc154-xn10_SN50",
                           OUT_1 => "01_PushButton"."SE01+NA1023-S1_PB",
                           OUT_2 => "01_PushButton"."SE01+NA1024-S1_PB",
                           OUT_3 => "01_PushButton"."SE01+NA1025-S1_PB",
                           OUT_4 => "01_PushButton"."SE01+NA1026-S1_PB");
END_REGION

REGION Network 13: 50.023 | n0023-uc154-xn10_SN50 [2]
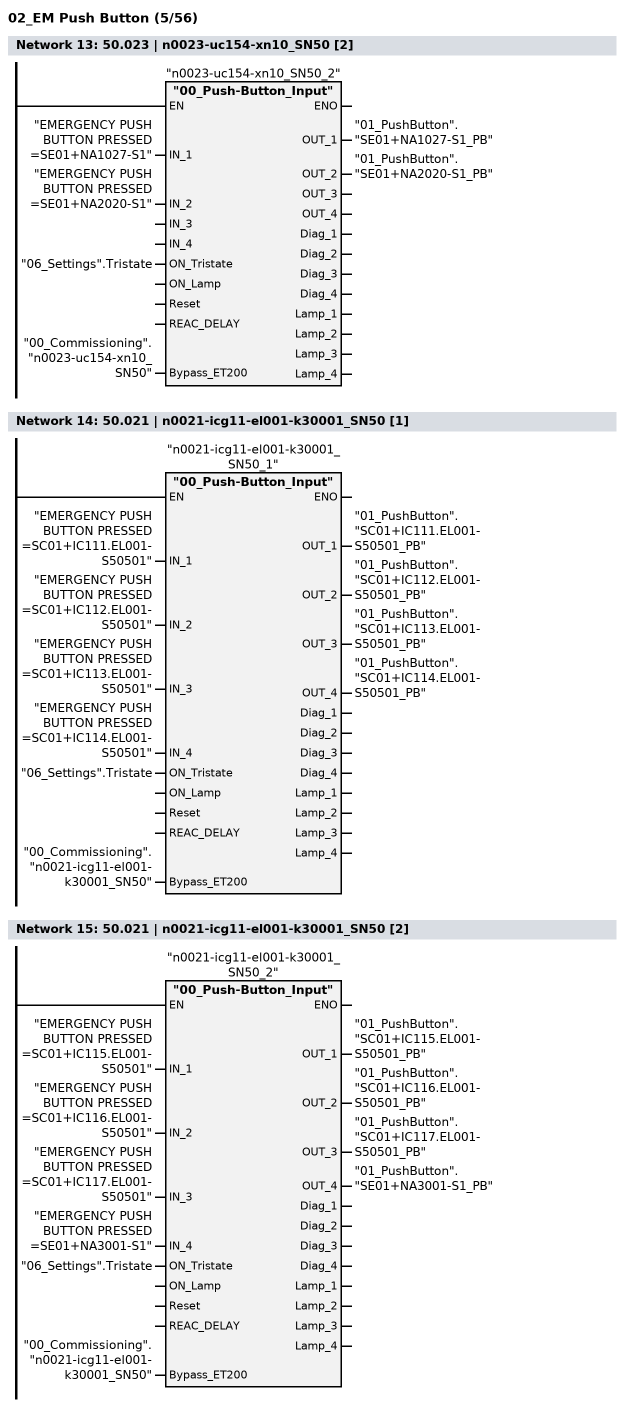
   RUNG wire#powerrail
      "n0023-uc154-xn10_SN50_2"(IN_1 := "EMERGENCY PUSH BUTTON PRESSED =SE01+NA1027-S1", IN_2 := "EMERGENCY PUSH BUTTON PRESSED =SE01+NA2020-S1", IN_3 :=, IN_4 :=, ON_Tristate := "06_Settings".Tristate, ON_Lamp :=, Reset :=, REAC_DELAY :=, Bypass_ET200 := "00_Commissioning"."n0023-uc154-xn10_SN50", OUT_1 => "01_PushButton"."SE01+NA1027-S1_PB", OUT_2 => "01_PushButton"."SE01+NA2020-S1_PB", OUT_3 =>, OUT_4 =>, Diag_1 =>, Diag_2 =>, Diag_3 =>, Diag_4 =>, Lamp_1 =>, Lamp_2 =>, Lamp_3 =>, Lamp_4 =>)
   END_RUNG
   // the same network as SCL:
   "n0023-uc154-xn10_SN50_2"(IN_1 := "EMERGENCY PUSH BUTTON PRESSED =SE01+NA1027-S1",   // "00_Push-Button_Input"
                           IN_2 := "EMERGENCY PUSH BUTTON PRESSED =SE01+NA2020-S1",
                           ON_Tristate := "06_Settings".Tristate,
                           Bypass_ET200 := "00_Commissioning"."n0023-uc154-xn10_SN50",
                           OUT_1 => "01_PushButton"."SE01+NA1027-S1_PB",
                           OUT_2 => "01_PushButton"."SE01+NA2020-S1_PB");
END_REGION

REGION Network 14: 50.021 | n0021-icg11-el001-k30001_SN50 [1]
   RUNG wire#powerrail
      "n0021-icg11-el001-k30001_SN50_1"(IN_1 := "EMERGENCY PUSH BUTTON PRESSED =SC01+IC111.EL001-S50501", IN_2 := "EMERGENCY PUSH BUTTON PRESSED =SC01+IC112.EL001-S50501", IN_3 := "EMERGENCY PUSH BUTTON PRESSED =SC01+IC113.EL001-S50501", IN_4 := "EMERGENCY PUSH BUTTON PRESSED =SC01+IC114.EL001-S50501", ON_Tristate := "06_Settings".Tristate, ON_Lamp :=, Reset :=, REAC_DELAY :=, Bypass_ET200 := "00_Commissioning"."n0021-icg11-el001-k30001_SN50", OUT_1 => "01_PushButton"."SC01+IC111.EL001-S50501_PB", OUT_2 => "01_PushButton"."SC01+IC112.EL001-S50501_PB", OUT_3 => "01_PushButton"."SC01+IC113.EL001-S50501_PB", OUT_4 => "01_PushButton"."SC01+IC114.EL001-S50501_PB", Diag_1 =>, Diag_2 =>, Diag_3 =>, Diag_4 =>, Lamp_1 =>, Lamp_2 =>, Lamp_3 =>, Lamp_4 =>)
   END_RUNG
   // the same network as SCL:
   "n0021-icg11-el001-k30001_SN50_1"(IN_1 := "EMERGENCY PUSH BUTTON PRESSED =SC01+IC111.EL001-S50501",   // "00_Push-Button_Input"
                           IN_2 := "EMERGENCY PUSH BUTTON PRESSED =SC01+IC112.EL001-S50501",
                           IN_3 := "EMERGENCY PUSH BUTTON PRESSED =SC01+IC113.EL001-S50501",
                           IN_4 := "EMERGENCY PUSH BUTTON PRESSED =SC01+IC114.EL001-S50501",
                           ON_Tristate := "06_Settings".Tristate,
                           Bypass_ET200 := "00_Commissioning"."n0021-icg11-el001-k30001_SN50",
                           OUT_1 => "01_PushButton"."SC01+IC111.EL001-S50501_PB",
                           OUT_2 => "01_PushButton"."SC01+IC112.EL001-S50501_PB",
                           OUT_3 => "01_PushButton"."SC01+IC113.EL001-S50501_PB",
                           OUT_4 => "01_PushButton"."SC01+IC114.EL001-S50501_PB");
END_REGION

REGION Network 15: 50.021 | n0021-icg11-el001-k30001_SN50 [2]
   RUNG wire#powerrail
      "n0021-icg11-el001-k30001_SN50_2"(IN_1 := "EMERGENCY PUSH BUTTON PRESSED =SC01+IC115.EL001-S50501", IN_2 := "EMERGENCY PUSH BUTTON PRESSED =SC01+IC116.EL001-S50501", IN_3 := "EMERGENCY PUSH BUTTON PRESSED =SC01+IC117.EL001-S50501", IN_4 := "EMERGENCY PUSH BUTTON PRESSED =SE01+NA3001-S1", ON_Tristate := "06_Settings".Tristate, ON_Lamp :=, Reset :=, REAC_DELAY :=, Bypass_ET200 := "00_Commissioning"."n0021-icg11-el001-k30001_SN50", OUT_1 => "01_PushButton"."SC01+IC115.EL001-S50501_PB", OUT_2 => "01_PushButton"."SC01+IC116.EL001-S50501_PB", OUT_3 => "01_PushButton"."SC01+IC117.EL001-S50501_PB", OUT_4 => "01_PushButton"."SE01+NA3001-S1_PB", Diag_1 =>, Diag_2 =>, Diag_3 =>, Diag_4 =>, Lamp_1 =>, Lamp_2 =>, Lamp_3 =>, Lamp_4 =>)
   END_RUNG
   // the same network as SCL:
   "n0021-icg11-el001-k30001_SN50_2"(IN_1 := "EMERGENCY PUSH BUTTON PRESSED =SC01+IC115.EL001-S50501",   // "00_Push-Button_Input"
                           IN_2 := "EMERGENCY PUSH BUTTON PRESSED =SC01+IC116.EL001-S50501",
                           IN_3 := "EMERGENCY PUSH BUTTON PRESSED =SC01+IC117.EL001-S50501",
                           IN_4 := "EMERGENCY PUSH BUTTON PRESSED =SE01+NA3001-S1",
                           ON_Tristate := "06_Settings".Tristate,
                           Bypass_ET200 := "00_Commissioning"."n0021-icg11-el001-k30001_SN50",
                           OUT_1 => "01_PushButton"."SC01+IC115.EL001-S50501_PB",
                           OUT_2 => "01_PushButton"."SC01+IC116.EL001-S50501_PB",
                           OUT_3 => "01_PushButton"."SC01+IC117.EL001-S50501_PB",
                           OUT_4 => "01_PushButton"."SE01+NA3001-S1_PB");
END_REGION

REGION Network 16: 50.021 | n0021-icg11-el001-k30001_SN50 [3]
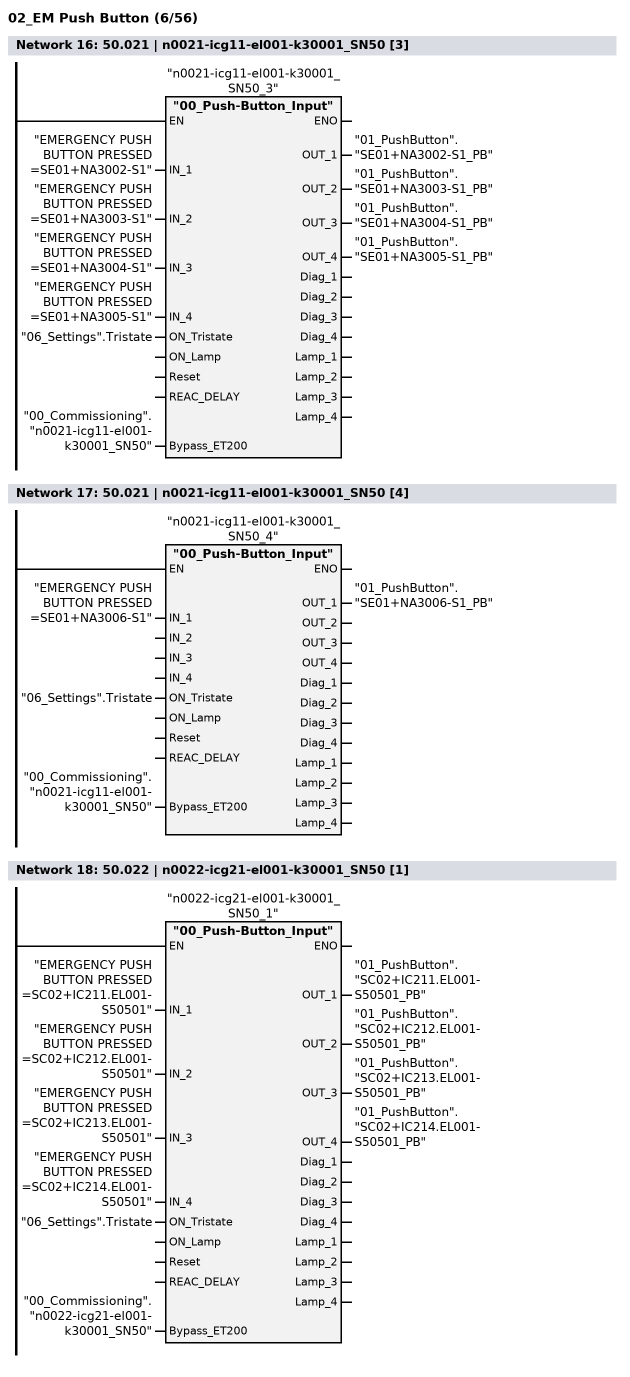
   RUNG wire#powerrail
      "n0021-icg11-el001-k30001_SN50_3"(IN_1 := "EMERGENCY PUSH BUTTON PRESSED =SE01+NA3002-S1", IN_2 := "EMERGENCY PUSH BUTTON PRESSED =SE01+NA3003-S1", IN_3 := "EMERGENCY PUSH BUTTON PRESSED =SE01+NA3004-S1", IN_4 := "EMERGENCY PUSH BUTTON PRESSED =SE01+NA3005-S1", ON_Tristate := "06_Settings".Tristate, ON_Lamp :=, Reset :=, REAC_DELAY :=, Bypass_ET200 := "00_Commissioning"."n0021-icg11-el001-k30001_SN50", OUT_1 => "01_PushButton"."SE01+NA3002-S1_PB", OUT_2 => "01_PushButton"."SE01+NA3003-S1_PB", OUT_3 => "01_PushButton"."SE01+NA3004-S1_PB", OUT_4 => "01_PushButton"."SE01+NA3005-S1_PB", Diag_1 =>, Diag_2 =>, Diag_3 =>, Diag_4 =>, Lamp_1 =>, Lamp_2 =>, Lamp_3 =>, Lamp_4 =>)
   END_RUNG
   // the same network as SCL:
   "n0021-icg11-el001-k30001_SN50_3"(IN_1 := "EMERGENCY PUSH BUTTON PRESSED =SE01+NA3002-S1",   // "00_Push-Button_Input"
                           IN_2 := "EMERGENCY PUSH BUTTON PRESSED =SE01+NA3003-S1",
                           IN_3 := "EMERGENCY PUSH BUTTON PRESSED =SE01+NA3004-S1",
                           IN_4 := "EMERGENCY PUSH BUTTON PRESSED =SE01+NA3005-S1",
                           ON_Tristate := "06_Settings".Tristate,
                           Bypass_ET200 := "00_Commissioning"."n0021-icg11-el001-k30001_SN50",
                           OUT_1 => "01_PushButton"."SE01+NA3002-S1_PB",
                           OUT_2 => "01_PushButton"."SE01+NA3003-S1_PB",
                           OUT_3 => "01_PushButton"."SE01+NA3004-S1_PB",
                           OUT_4 => "01_PushButton"."SE01+NA3005-S1_PB");
END_REGION

REGION Network 17: 50.021 | n0021-icg11-el001-k30001_SN50 [4]
   RUNG wire#powerrail
      "n0021-icg11-el001-k30001_SN50_4"(IN_1 := "EMERGENCY PUSH BUTTON PRESSED =SE01+NA3006-S1", IN_2 :=, IN_3 :=, IN_4 :=, ON_Tristate := "06_Settings".Tristate, ON_Lamp :=, Reset :=, REAC_DELAY :=, Bypass_ET200 := "00_Commissioning"."n0021-icg11-el001-k30001_SN50", OUT_1 => "01_PushButton"."SE01+NA3006-S1_PB", OUT_2 =>, OUT_3 =>, OUT_4 =>, Diag_1 =>, Diag_2 =>, Diag_3 =>, Diag_4 =>, Lamp_1 =>, Lamp_2 =>, Lamp_3 =>, Lamp_4 =>)
   END_RUNG
   // the same network as SCL:
   "n0021-icg11-el001-k30001_SN50_4"(IN_1 := "EMERGENCY PUSH BUTTON PRESSED =SE01+NA3006-S1",   // "00_Push-Button_Input"
                           ON_Tristate := "06_Settings".Tristate,
                           Bypass_ET200 := "00_Commissioning"."n0021-icg11-el001-k30001_SN50",
                           OUT_1 => "01_PushButton"."SE01+NA3006-S1_PB");
END_REGION

REGION Network 18: 50.022 | n0022-icg21-el001-k30001_SN50 [1]
   RUNG wire#powerrail
      "n0022-icg21-el001-k30001_SN50_1"(IN_1 := "EMERGENCY PUSH BUTTON PRESSED =SC02+IC211.EL001-S50501", IN_2 := "EMERGENCY PUSH BUTTON PRESSED =SC02+IC212.EL001-S50501", IN_3 := "EMERGENCY PUSH BUTTON PRESSED =SC02+IC213.EL001-S50501", IN_4 := "EMERGENCY PUSH BUTTON PRESSED =SC02+IC214.EL001-S50501", ON_Tristate := "06_Settings".Tristate, ON_Lamp :=, Reset :=, REAC_DELAY :=, Bypass_ET200 := "00_Commissioning"."n0022-icg21-el001-k30001_SN50", OUT_1 => "01_PushButton"."SC02+IC211.EL001-S50501_PB", OUT_2 => "01_PushButton"."SC02+IC212.EL001-S50501_PB", OUT_3 => "01_PushButton"."SC02+IC213.EL001-S50501_PB", OUT_4 => "01_PushButton"."SC02+IC214.EL001-S50501_PB", Diag_1 =>, Diag_2 =>, Diag_3 =>, Diag_4 =>, Lamp_1 =>, Lamp_2 =>, Lamp_3 =>, Lamp_4 =>)
   END_RUNG
   // the same network as SCL:
   "n0022-icg21-el001-k30001_SN50_1"(IN_1 := "EMERGENCY PUSH BUTTON PRESSED =SC02+IC211.EL001-S50501",   // "00_Push-Button_Input"
                           IN_2 := "EMERGENCY PUSH BUTTON PRESSED =SC02+IC212.EL001-S50501",
                           IN_3 := "EMERGENCY PUSH BUTTON PRESSED =SC02+IC213.EL001-S50501",
                           IN_4 := "EMERGENCY PUSH BUTTON PRESSED =SC02+IC214.EL001-S50501",
                           ON_Tristate := "06_Settings".Tristate,
                           Bypass_ET200 := "00_Commissioning"."n0022-icg21-el001-k30001_SN50",
                           OUT_1 => "01_PushButton"."SC02+IC211.EL001-S50501_PB",
                           OUT_2 => "01_PushButton"."SC02+IC212.EL001-S50501_PB",
                           OUT_3 => "01_PushButton"."SC02+IC213.EL001-S50501_PB",
                           OUT_4 => "01_PushButton"."SC02+IC214.EL001-S50501_PB");
END_REGION

REGION Network 19: 50.022 | n0022-icg21-el001-k30001_SN50 [2]
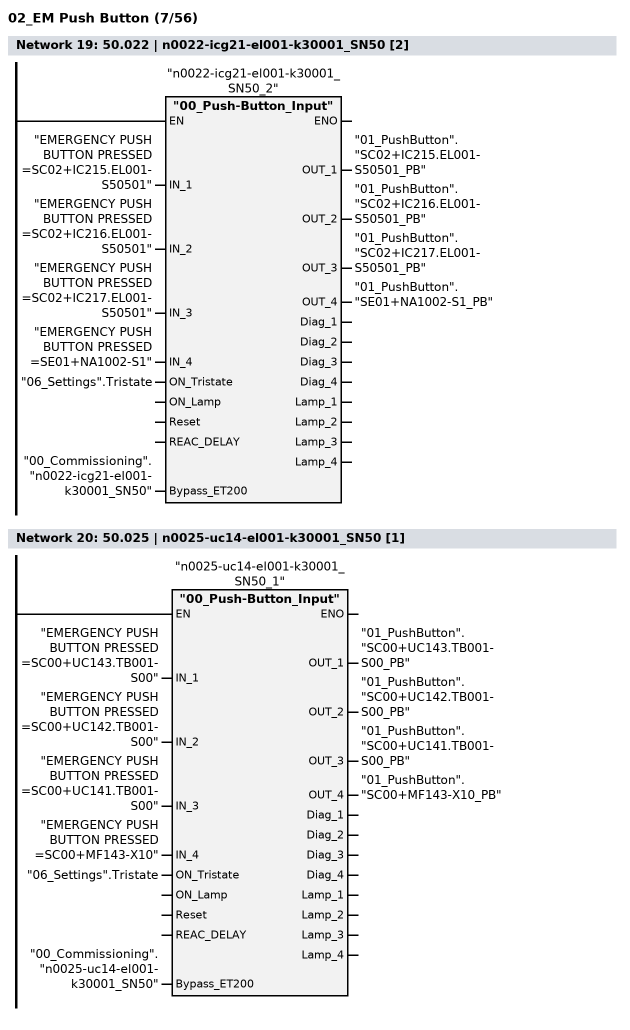
   RUNG wire#powerrail
      "n0022-icg21-el001-k30001_SN50_2"(IN_1 := "EMERGENCY PUSH BUTTON PRESSED =SC02+IC215.EL001-S50501", IN_2 := "EMERGENCY PUSH BUTTON PRESSED =SC02+IC216.EL001-S50501", IN_3 := "EMERGENCY PUSH BUTTON PRESSED =SC02+IC217.EL001-S50501", IN_4 := "EMERGENCY PUSH BUTTON PRESSED =SE01+NA1002-S1", ON_Tristate := "06_Settings".Tristate, ON_Lamp :=, Reset :=, REAC_DELAY :=, Bypass_ET200 := "00_Commissioning"."n0022-icg21-el001-k30001_SN50", OUT_1 => "01_PushButton"."SC02+IC215.EL001-S50501_PB", OUT_2 => "01_PushButton"."SC02+IC216.EL001-S50501_PB", OUT_3 => "01_PushButton"."SC02+IC217.EL001-S50501_PB", OUT_4 => "01_PushButton"."SE01+NA1002-S1_PB", Diag_1 =>, Diag_2 =>, Diag_3 =>, Diag_4 =>, Lamp_1 =>, Lamp_2 =>, Lamp_3 =>, Lamp_4 =>)
   END_RUNG
   // the same network as SCL:
   "n0022-icg21-el001-k30001_SN50_2"(IN_1 := "EMERGENCY PUSH BUTTON PRESSED =SC02+IC215.EL001-S50501",   // "00_Push-Button_Input"
                           IN_2 := "EMERGENCY PUSH BUTTON PRESSED =SC02+IC216.EL001-S50501",
                           IN_3 := "EMERGENCY PUSH BUTTON PRESSED =SC02+IC217.EL001-S50501",
                           IN_4 := "EMERGENCY PUSH BUTTON PRESSED =SE01+NA1002-S1",
                           ON_Tristate := "06_Settings".Tristate,
                           Bypass_ET200 := "00_Commissioning"."n0022-icg21-el001-k30001_SN50",
                           OUT_1 => "01_PushButton"."SC02+IC215.EL001-S50501_PB",
                           OUT_2 => "01_PushButton"."SC02+IC216.EL001-S50501_PB",
                           OUT_3 => "01_PushButton"."SC02+IC217.EL001-S50501_PB",
                           OUT_4 => "01_PushButton"."SE01+NA1002-S1_PB");
END_REGION

REGION Network 20: 50.025 | n0025-uc14-el001-k30001_SN50 [1]
   RUNG wire#powerrail
      "n0025-uc14-el001-k30001_SN50_1"(IN_1 := "EMERGENCY PUSH BUTTON PRESSED =SC00+UC143.TB001-S00", IN_2 := "EMERGENCY PUSH BUTTON PRESSED =SC00+UC142.TB001-S00", IN_3 := "EMERGENCY PUSH BUTTON PRESSED =SC00+UC141.TB001-S00", IN_4 := "EMERGENCY PUSH BUTTON PRESSED =SC00+MF143-X10", ON_Tristate := "06_Settings".Tristate, ON_Lamp :=, Reset :=, REAC_DELAY :=, Bypass_ET200 := "00_Commissioning"."n0025-uc14-el001-k30001_SN50", OUT_1 => "01_PushButton"."SC00+UC143.TB001-S00_PB", OUT_2 => "01_PushButton"."SC00+UC142.TB001-S00_PB", OUT_3 => "01_PushButton"."SC00+UC141.TB001-S00_PB", OUT_4 => "01_PushButton"."SC00+MF143-X10_PB", Diag_1 =>, Diag_2 =>, Diag_3 =>, Diag_4 =>, Lamp_1 =>, Lamp_2 =>, Lamp_3 =>, Lamp_4 =>)
   END_RUNG
   // the same network as SCL:
   "n0025-uc14-el001-k30001_SN50_1"(IN_1 := "EMERGENCY PUSH BUTTON PRESSED =SC00+UC143.TB001-S00",   // "00_Push-Button_Input"
                           IN_2 := "EMERGENCY PUSH BUTTON PRESSED =SC00+UC142.TB001-S00",
                           IN_3 := "EMERGENCY PUSH BUTTON PRESSED =SC00+UC141.TB001-S00",
                           IN_4 := "EMERGENCY PUSH BUTTON PRESSED =SC00+MF143-X10",
                           ON_Tristate := "06_Settings".Tristate,
                           Bypass_ET200 := "00_Commissioning"."n0025-uc14-el001-k30001_SN50",
                           OUT_1 => "01_PushButton"."SC00+UC143.TB001-S00_PB",
                           OUT_2 => "01_PushButton"."SC00+UC142.TB001-S00_PB",
                           OUT_3 => "01_PushButton"."SC00+UC141.TB001-S00_PB",
                           OUT_4 => "01_PushButton"."SC00+MF143-X10_PB");
END_REGION

REGION Network 21: 50.025 | n0025-uc14-el001-k30001_SN50 [2]
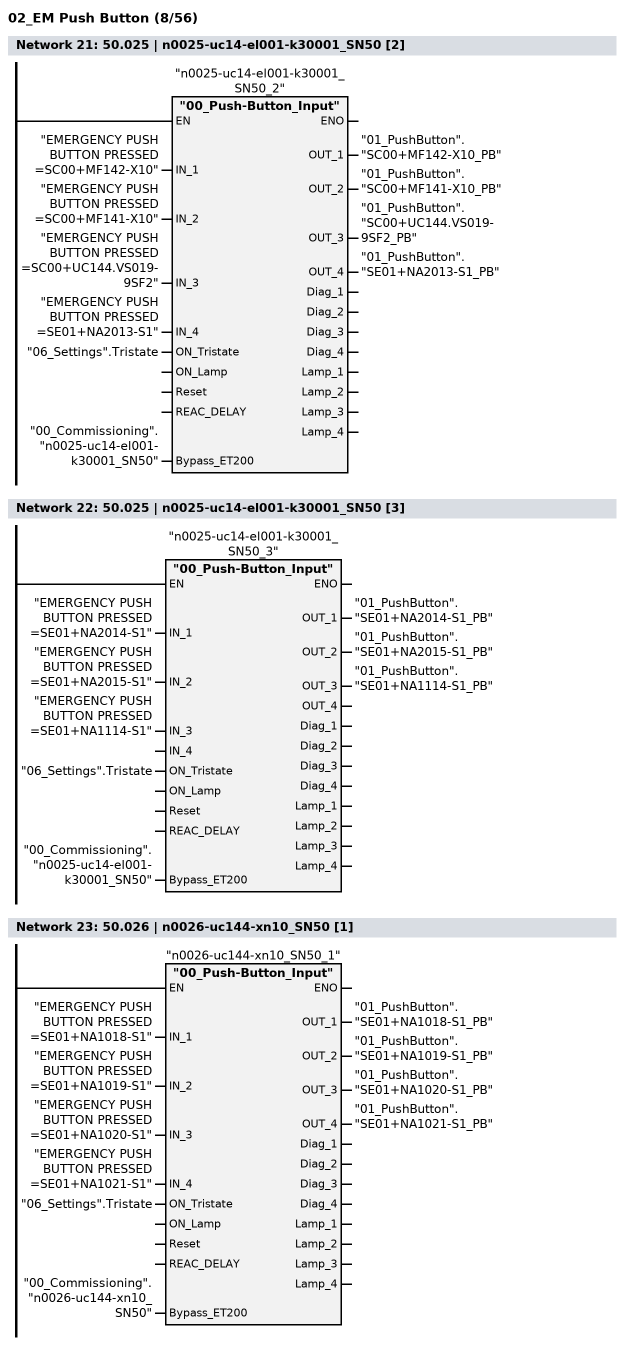
   RUNG wire#powerrail
      "n0025-uc14-el001-k30001_SN50_2"(IN_1 := "EMERGENCY PUSH BUTTON PRESSED =SC00+MF142-X10", IN_2 := "EMERGENCY PUSH BUTTON PRESSED =SC00+MF141-X10", IN_3 := "EMERGENCY PUSH BUTTON PRESSED =SC00+UC144.VS019-9SF2", IN_4 := "EMERGENCY PUSH BUTTON PRESSED =SE01+NA2013-S1", ON_Tristate := "06_Settings".Tristate, ON_Lamp :=, Reset :=, REAC_DELAY :=, Bypass_ET200 := "00_Commissioning"."n0025-uc14-el001-k30001_SN50", OUT_1 => "01_PushButton"."SC00+MF142-X10_PB", OUT_2 => "01_PushButton"."SC00+MF141-X10_PB", OUT_3 => "01_PushButton"."SC00+UC144.VS019-9SF2_PB", OUT_4 => "01_PushButton"."SE01+NA2013-S1_PB", Diag_1 =>, Diag_2 =>, Diag_3 =>, Diag_4 =>, Lamp_1 =>, Lamp_2 =>, Lamp_3 =>, Lamp_4 =>)
   END_RUNG
   // the same network as SCL:
   "n0025-uc14-el001-k30001_SN50_2"(IN_1 := "EMERGENCY PUSH BUTTON PRESSED =SC00+MF142-X10",   // "00_Push-Button_Input"
                           IN_2 := "EMERGENCY PUSH BUTTON PRESSED =SC00+MF141-X10",
                           IN_3 := "EMERGENCY PUSH BUTTON PRESSED =SC00+UC144.VS019-9SF2",
                           IN_4 := "EMERGENCY PUSH BUTTON PRESSED =SE01+NA2013-S1",
                           ON_Tristate := "06_Settings".Tristate,
                           Bypass_ET200 := "00_Commissioning"."n0025-uc14-el001-k30001_SN50",
                           OUT_1 => "01_PushButton"."SC00+MF142-X10_PB",
                           OUT_2 => "01_PushButton"."SC00+MF141-X10_PB",
                           OUT_3 => "01_PushButton"."SC00+UC144.VS019-9SF2_PB",
                           OUT_4 => "01_PushButton"."SE01+NA2013-S1_PB");
END_REGION

REGION Network 22: 50.025 | n0025-uc14-el001-k30001_SN50 [3]
   RUNG wire#powerrail
      "n0025-uc14-el001-k30001_SN50_3"(IN_1 := "EMERGENCY PUSH BUTTON PRESSED =SE01+NA2014-S1", IN_2 := "EMERGENCY PUSH BUTTON PRESSED =SE01+NA2015-S1", IN_3 := "EMERGENCY PUSH BUTTON PRESSED =SE01+NA1114-S1", IN_4 :=, ON_Tristate := "06_Settings".Tristate, ON_Lamp :=, Reset :=, REAC_DELAY :=, Bypass_ET200 := "00_Commissioning"."n0025-uc14-el001-k30001_SN50", OUT_1 => "01_PushButton"."SE01+NA2014-S1_PB", OUT_2 => "01_PushButton"."SE01+NA2015-S1_PB", OUT_3 => "01_PushButton"."SE01+NA1114-S1_PB", OUT_4 =>, Diag_1 =>, Diag_2 =>, Diag_3 =>, Diag_4 =>, Lamp_1 =>, Lamp_2 =>, Lamp_3 =>, Lamp_4 =>)
   END_RUNG
   // the same network as SCL:
   "n0025-uc14-el001-k30001_SN50_3"(IN_1 := "EMERGENCY PUSH BUTTON PRESSED =SE01+NA2014-S1",   // "00_Push-Button_Input"
                           IN_2 := "EMERGENCY PUSH BUTTON PRESSED =SE01+NA2015-S1",
                           IN_3 := "EMERGENCY PUSH BUTTON PRESSED =SE01+NA1114-S1",
                           ON_Tristate := "06_Settings".Tristate,
                           Bypass_ET200 := "00_Commissioning"."n0025-uc14-el001-k30001_SN50",
                           OUT_1 => "01_PushButton"."SE01+NA2014-S1_PB",
                           OUT_2 => "01_PushButton"."SE01+NA2015-S1_PB",
                           OUT_3 => "01_PushButton"."SE01+NA1114-S1_PB");
END_REGION

REGION Network 23: 50.026 | n0026-uc144-xn10_SN50 [1]
   RUNG wire#powerrail
      "n0026-uc144-xn10_SN50_1"(IN_1 := "EMERGENCY PUSH BUTTON PRESSED =SE01+NA1018-S1", IN_2 := "EMERGENCY PUSH BUTTON PRESSED =SE01+NA1019-S1", IN_3 := "EMERGENCY PUSH BUTTON PRESSED =SE01+NA1020-S1", IN_4 := "EMERGENCY PUSH BUTTON PRESSED =SE01+NA1021-S1", ON_Tristate := "06_Settings".Tristate, ON_Lamp :=, Reset :=, REAC_DELAY :=, Bypass_ET200 := "00_Commissioning"."n0026-uc144-xn10_SN50", OUT_1 => "01_PushButton"."SE01+NA1018-S1_PB", OUT_2 => "01_PushButton"."SE01+NA1019-S1_PB", OUT_3 => "01_PushButton"."SE01+NA1020-S1_PB", OUT_4 => "01_PushButton"."SE01+NA1021-S1_PB", Diag_1 =>, Diag_2 =>, Diag_3 =>, Diag_4 =>, Lamp_1 =>, Lamp_2 =>, Lamp_3 =>, Lamp_4 =>)
   END_RUNG
   // the same network as SCL:
   "n0026-uc144-xn10_SN50_1"(IN_1 := "EMERGENCY PUSH BUTTON PRESSED =SE01+NA1018-S1",   // "00_Push-Button_Input"
                           IN_2 := "EMERGENCY PUSH BUTTON PRESSED =SE01+NA1019-S1",
                           IN_3 := "EMERGENCY PUSH BUTTON PRESSED =SE01+NA1020-S1",
                           IN_4 := "EMERGENCY PUSH BUTTON PRESSED =SE01+NA1021-S1",
                           ON_Tristate := "06_Settings".Tristate,
                           Bypass_ET200 := "00_Commissioning"."n0026-uc144-xn10_SN50",
                           OUT_1 => "01_PushButton"."SE01+NA1018-S1_PB",
                           OUT_2 => "01_PushButton"."SE01+NA1019-S1_PB",
                           OUT_3 => "01_PushButton"."SE01+NA1020-S1_PB",
                           OUT_4 => "01_PushButton"."SE01+NA1021-S1_PB");
END_REGION

REGION Network 24: 50.026 | n0026-uc144-xn10_SN50 [2]
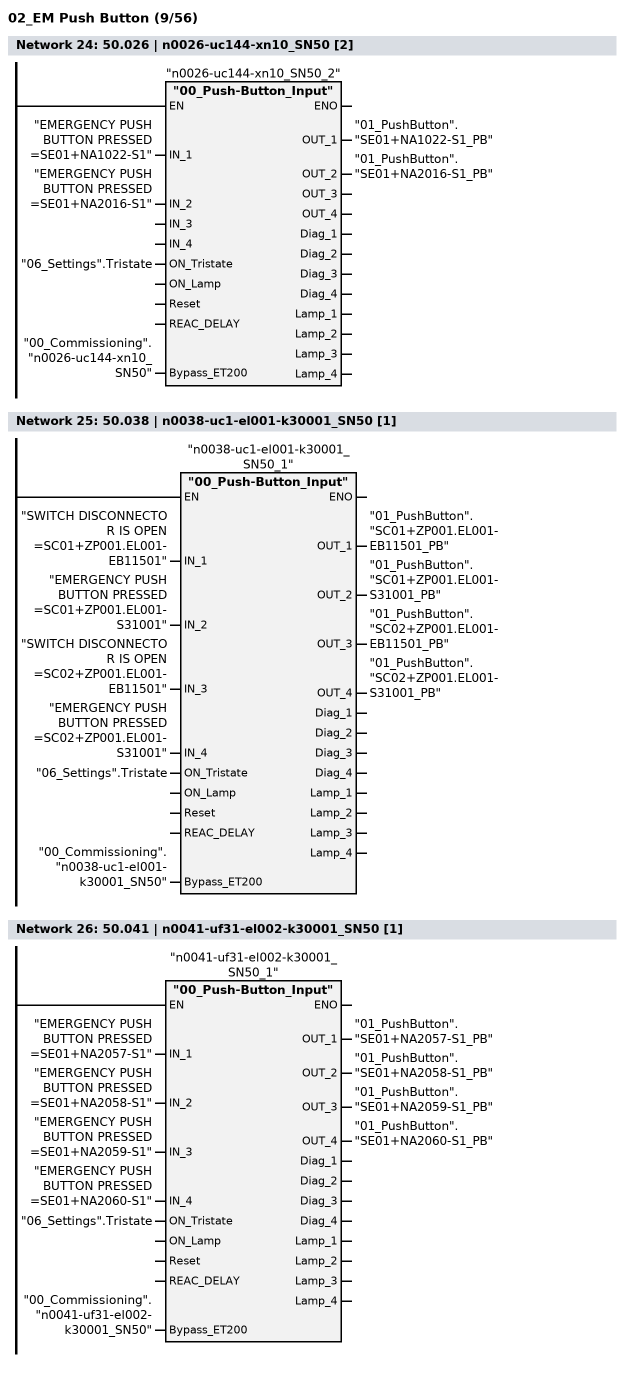
   RUNG wire#powerrail
      "n0026-uc144-xn10_SN50_2"(IN_1 := "EMERGENCY PUSH BUTTON PRESSED =SE01+NA1022-S1", IN_2 := "EMERGENCY PUSH BUTTON PRESSED =SE01+NA2016-S1", IN_3 :=, IN_4 :=, ON_Tristate := "06_Settings".Tristate, ON_Lamp :=, Reset :=, REAC_DELAY :=, Bypass_ET200 := "00_Commissioning"."n0026-uc144-xn10_SN50", OUT_1 => "01_PushButton"."SE01+NA1022-S1_PB", OUT_2 => "01_PushButton"."SE01+NA2016-S1_PB", OUT_3 =>, OUT_4 =>, Diag_1 =>, Diag_2 =>, Diag_3 =>, Diag_4 =>, Lamp_1 =>, Lamp_2 =>, Lamp_3 =>, Lamp_4 =>)
   END_RUNG
   // the same network as SCL:
   "n0026-uc144-xn10_SN50_2"(IN_1 := "EMERGENCY PUSH BUTTON PRESSED =SE01+NA1022-S1",   // "00_Push-Button_Input"
                           IN_2 := "EMERGENCY PUSH BUTTON PRESSED =SE01+NA2016-S1",
                           ON_Tristate := "06_Settings".Tristate,
                           Bypass_ET200 := "00_Commissioning"."n0026-uc144-xn10_SN50",
                           OUT_1 => "01_PushButton"."SE01+NA1022-S1_PB",
                           OUT_2 => "01_PushButton"."SE01+NA2016-S1_PB");
END_REGION

REGION Network 25: 50.038 | n0038-uc1-el001-k30001_SN50 [1]
   RUNG wire#powerrail
      "n0038-uc1-el001-k30001_SN50_1"(IN_1 := "SWITCH DISCONNECTOR IS OPEN =SC01+ZP001.EL001-EB11501", IN_2 := "EMERGENCY PUSH BUTTON PRESSED =SC01+ZP001.EL001-S31001", IN_3 := "SWITCH DISCONNECTOR IS OPEN =SC02+ZP001.EL001-EB11501", IN_4 := "EMERGENCY PUSH BUTTON PRESSED =SC02+ZP001.EL001-S31001", ON_Tristate := "06_Settings".Tristate, ON_Lamp :=, Reset :=, REAC_DELAY :=, Bypass_ET200 := "00_Commissioning"."n0038-uc1-el001-k30001_SN50", OUT_1 => "01_PushButton"."SC01+ZP001.EL001-EB11501_PB", OUT_2 => "01_PushButton"."SC01+ZP001.EL001-S31001_PB", OUT_3 => "01_PushButton"."SC02+ZP001.EL001-EB11501_PB", OUT_4 => "01_PushButton"."SC02+ZP001.EL001-S31001_PB", Diag_1 =>, Diag_2 =>, Diag_3 =>, Diag_4 =>, Lamp_1 =>, Lamp_2 =>, Lamp_3 =>, Lamp_4 =>)
   END_RUNG
   // the same network as SCL:
   "n0038-uc1-el001-k30001_SN50_1"(IN_1 := "SWITCH DISCONNECTOR IS OPEN =SC01+ZP001.EL001-EB11501",   // "00_Push-Button_Input"
                           IN_2 := "EMERGENCY PUSH BUTTON PRESSED =SC01+ZP001.EL001-S31001",
                           IN_3 := "SWITCH DISCONNECTOR IS OPEN =SC02+ZP001.EL001-EB11501",
                           IN_4 := "EMERGENCY PUSH BUTTON PRESSED =SC02+ZP001.EL001-S31001",
                           ON_Tristate := "06_Settings".Tristate,
                           Bypass_ET200 := "00_Commissioning"."n0038-uc1-el001-k30001_SN50",
                           OUT_1 => "01_PushButton"."SC01+ZP001.EL001-EB11501_PB",
                           OUT_2 => "01_PushButton"."SC01+ZP001.EL001-S31001_PB",
                           OUT_3 => "01_PushButton"."SC02+ZP001.EL001-EB11501_PB",
                           OUT_4 => "01_PushButton"."SC02+ZP001.EL001-S31001_PB");
END_REGION

REGION Network 26: 50.041 | n0041-uf31-el002-k30001_SN50 [1]
   RUNG wire#powerrail
      "n0041-uf31-el002-k30001_SN50_1"(IN_1 := "EMERGENCY PUSH BUTTON PRESSED =SE01+NA2057-S1", IN_2 := "EMERGENCY PUSH BUTTON PRESSED =SE01+NA2058-S1", IN_3 := "EMERGENCY PUSH BUTTON PRESSED =SE01+NA2059-S1", IN_4 := "EMERGENCY PUSH BUTTON PRESSED =SE01+NA2060-S1", ON_Tristate := "06_Settings".Tristate, ON_Lamp :=, Reset :=, REAC_DELAY :=, Bypass_ET200 := "00_Commissioning"."n0041-uf31-el002-k30001_SN50", OUT_1 => "01_PushButton"."SE01+NA2057-S1_PB", OUT_2 => "01_PushButton"."SE01+NA2058-S1_PB", OUT_3 => "01_PushButton"."SE01+NA2059-S1_PB", OUT_4 => "01_PushButton"."SE01+NA2060-S1_PB", Diag_1 =>, Diag_2 =>, Diag_3 =>, Diag_4 =>, Lamp_1 =>, Lamp_2 =>, Lamp_3 =>, Lamp_4 =>)
   END_RUNG
   // the same network as SCL:
   "n0041-uf31-el002-k30001_SN50_1"(IN_1 := "EMERGENCY PUSH BUTTON PRESSED =SE01+NA2057-S1",   // "00_Push-Button_Input"
                           IN_2 := "EMERGENCY PUSH BUTTON PRESSED =SE01+NA2058-S1",
                           IN_3 := "EMERGENCY PUSH BUTTON PRESSED =SE01+NA2059-S1",
                           IN_4 := "EMERGENCY PUSH BUTTON PRESSED =SE01+NA2060-S1",
                           ON_Tristate := "06_Settings".Tristate,
                           Bypass_ET200 := "00_Commissioning"."n0041-uf31-el002-k30001_SN50",
                           OUT_1 => "01_PushButton"."SE01+NA2057-S1_PB",
                           OUT_2 => "01_PushButton"."SE01+NA2058-S1_PB",
                           OUT_3 => "01_PushButton"."SE01+NA2059-S1_PB",
                           OUT_4 => "01_PushButton"."SE01+NA2060-S1_PB");
END_REGION

REGION Network 27: 50.044 | n0044-ct1-el001-k30001_SN50 [1]
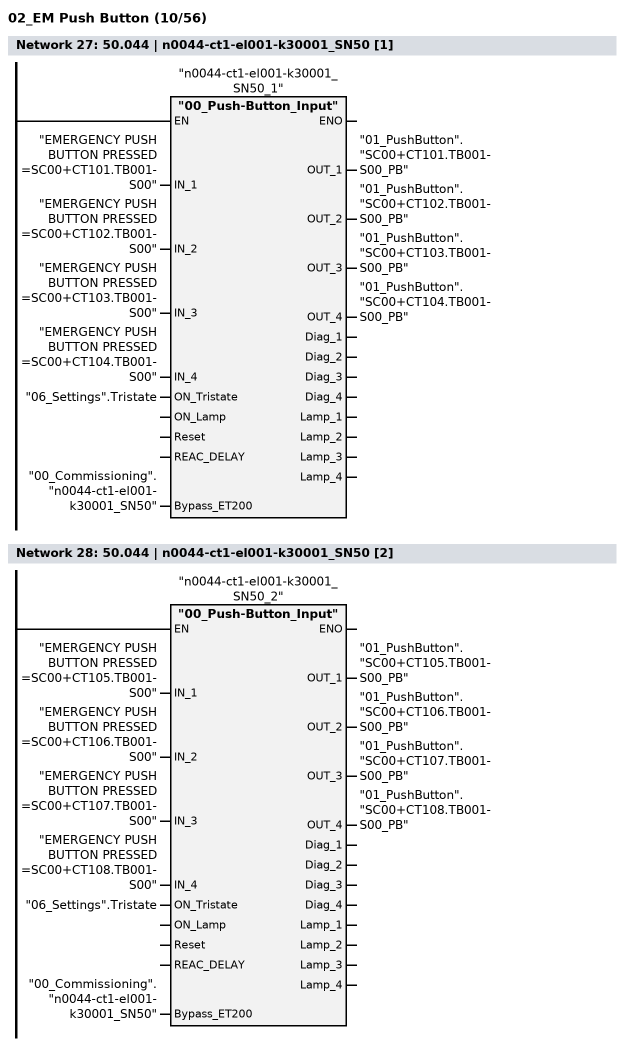
   RUNG wire#powerrail
      "n0044-ct1-el001-k30001_SN50_1"(IN_1 := "EMERGENCY PUSH BUTTON PRESSED =SC00+CT101.TB001-S00", IN_2 := "EMERGENCY PUSH BUTTON PRESSED =SC00+CT102.TB001-S00", IN_3 := "EMERGENCY PUSH BUTTON PRESSED =SC00+CT103.TB001-S00", IN_4 := "EMERGENCY PUSH BUTTON PRESSED =SC00+CT104.TB001-S00", ON_Tristate := "06_Settings".Tristate, ON_Lamp :=, Reset :=, REAC_DELAY :=, Bypass_ET200 := "00_Commissioning"."n0044-ct1-el001-k30001_SN50", OUT_1 => "01_PushButton"."SC00+CT101.TB001-S00_PB", OUT_2 => "01_PushButton"."SC00+CT102.TB001-S00_PB", OUT_3 => "01_PushButton"."SC00+CT103.TB001-S00_PB", OUT_4 => "01_PushButton"."SC00+CT104.TB001-S00_PB", Diag_1 =>, Diag_2 =>, Diag_3 =>, Diag_4 =>, Lamp_1 =>, Lamp_2 =>, Lamp_3 =>, Lamp_4 =>)
   END_RUNG
   // the same network as SCL:
   "n0044-ct1-el001-k30001_SN50_1"(IN_1 := "EMERGENCY PUSH BUTTON PRESSED =SC00+CT101.TB001-S00",   // "00_Push-Button_Input"
                           IN_2 := "EMERGENCY PUSH BUTTON PRESSED =SC00+CT102.TB001-S00",
                           IN_3 := "EMERGENCY PUSH BUTTON PRESSED =SC00+CT103.TB001-S00",
                           IN_4 := "EMERGENCY PUSH BUTTON PRESSED =SC00+CT104.TB001-S00",
                           ON_Tristate := "06_Settings".Tristate,
                           Bypass_ET200 := "00_Commissioning"."n0044-ct1-el001-k30001_SN50",
                           OUT_1 => "01_PushButton"."SC00+CT101.TB001-S00_PB",
                           OUT_2 => "01_PushButton"."SC00+CT102.TB001-S00_PB",
                           OUT_3 => "01_PushButton"."SC00+CT103.TB001-S00_PB",
                           OUT_4 => "01_PushButton"."SC00+CT104.TB001-S00_PB");
END_REGION

REGION Network 28: 50.044 | n0044-ct1-el001-k30001_SN50 [2]
   RUNG wire#powerrail
      "n0044-ct1-el001-k30001_SN50_2"(IN_1 := "EMERGENCY PUSH BUTTON PRESSED =SC00+CT105.TB001-S00", IN_2 := "EMERGENCY PUSH BUTTON PRESSED =SC00+CT106.TB001-S00", IN_3 := "EMERGENCY PUSH BUTTON PRESSED =SC00+CT107.TB001-S00", IN_4 := "EMERGENCY PUSH BUTTON PRESSED =SC00+CT108.TB001-S00", ON_Tristate := "06_Settings".Tristate, ON_Lamp :=, Reset :=, REAC_DELAY :=, Bypass_ET200 := "00_Commissioning"."n0044-ct1-el001-k30001_SN50", OUT_1 => "01_PushButton"."SC00+CT105.TB001-S00_PB", OUT_2 => "01_PushButton"."SC00+CT106.TB001-S00_PB", OUT_3 => "01_PushButton"."SC00+CT107.TB001-S00_PB", OUT_4 => "01_PushButton"."SC00+CT108.TB001-S00_PB", Diag_1 =>, Diag_2 =>, Diag_3 =>, Diag_4 =>, Lamp_1 =>, Lamp_2 =>, Lamp_3 =>, Lamp_4 =>)
   END_RUNG
   // the same network as SCL:
   "n0044-ct1-el001-k30001_SN50_2"(IN_1 := "EMERGENCY PUSH BUTTON PRESSED =SC00+CT105.TB001-S00",   // "00_Push-Button_Input"
                           IN_2 := "EMERGENCY PUSH BUTTON PRESSED =SC00+CT106.TB001-S00",
                           IN_3 := "EMERGENCY PUSH BUTTON PRESSED =SC00+CT107.TB001-S00",
                           IN_4 := "EMERGENCY PUSH BUTTON PRESSED =SC00+CT108.TB001-S00",
                           ON_Tristate := "06_Settings".Tristate,
                           Bypass_ET200 := "00_Commissioning"."n0044-ct1-el001-k30001_SN50",
                           OUT_1 => "01_PushButton"."SC00+CT105.TB001-S00_PB",
                           OUT_2 => "01_PushButton"."SC00+CT106.TB001-S00_PB",
                           OUT_3 => "01_PushButton"."SC00+CT107.TB001-S00_PB",
                           OUT_4 => "01_PushButton"."SC00+CT108.TB001-S00_PB");
END_REGION

REGION Network 29: 50.044 | n0044-ct1-el001-k30001_SN50 [3]
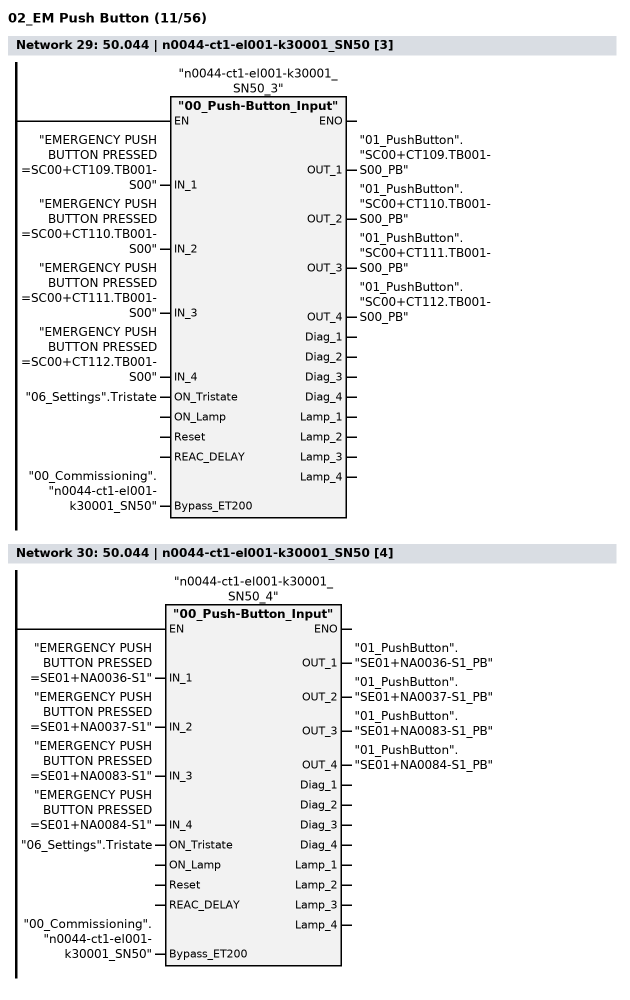
   RUNG wire#powerrail
      "n0044-ct1-el001-k30001_SN50_3"(IN_1 := "EMERGENCY PUSH BUTTON PRESSED =SC00+CT109.TB001-S00", IN_2 := "EMERGENCY PUSH BUTTON PRESSED =SC00+CT110.TB001-S00", IN_3 := "EMERGENCY PUSH BUTTON PRESSED =SC00+CT111.TB001-S00", IN_4 := "EMERGENCY PUSH BUTTON PRESSED =SC00+CT112.TB001-S00", ON_Tristate := "06_Settings".Tristate, ON_Lamp :=, Reset :=, REAC_DELAY :=, Bypass_ET200 := "00_Commissioning"."n0044-ct1-el001-k30001_SN50", OUT_1 => "01_PushButton"."SC00+CT109.TB001-S00_PB", OUT_2 => "01_PushButton"."SC00+CT110.TB001-S00_PB", OUT_3 => "01_PushButton"."SC00+CT111.TB001-S00_PB", OUT_4 => "01_PushButton"."SC00+CT112.TB001-S00_PB", Diag_1 =>, Diag_2 =>, Diag_3 =>, Diag_4 =>, Lamp_1 =>, Lamp_2 =>, Lamp_3 =>, Lamp_4 =>)
   END_RUNG
   // the same network as SCL:
   "n0044-ct1-el001-k30001_SN50_3"(IN_1 := "EMERGENCY PUSH BUTTON PRESSED =SC00+CT109.TB001-S00",   // "00_Push-Button_Input"
                           IN_2 := "EMERGENCY PUSH BUTTON PRESSED =SC00+CT110.TB001-S00",
                           IN_3 := "EMERGENCY PUSH BUTTON PRESSED =SC00+CT111.TB001-S00",
                           IN_4 := "EMERGENCY PUSH BUTTON PRESSED =SC00+CT112.TB001-S00",
                           ON_Tristate := "06_Settings".Tristate,
                           Bypass_ET200 := "00_Commissioning"."n0044-ct1-el001-k30001_SN50",
                           OUT_1 => "01_PushButton"."SC00+CT109.TB001-S00_PB",
                           OUT_2 => "01_PushButton"."SC00+CT110.TB001-S00_PB",
                           OUT_3 => "01_PushButton"."SC00+CT111.TB001-S00_PB",
                           OUT_4 => "01_PushButton"."SC00+CT112.TB001-S00_PB");
END_REGION

REGION Network 30: 50.044 | n0044-ct1-el001-k30001_SN50 [4]
   RUNG wire#powerrail
      "n0044-ct1-el001-k30001_SN50_4"(IN_1 := "EMERGENCY PUSH BUTTON PRESSED =SE01+NA0036-S1", IN_2 := "EMERGENCY PUSH BUTTON PRESSED =SE01+NA0037-S1", IN_3 := "EMERGENCY PUSH BUTTON PRESSED =SE01+NA0083-S1", IN_4 := "EMERGENCY PUSH BUTTON PRESSED =SE01+NA0084-S1", ON_Tristate := "06_Settings".Tristate, ON_Lamp :=, Reset :=, REAC_DELAY :=, Bypass_ET200 := "00_Commissioning"."n0044-ct1-el001-k30001_SN50", OUT_1 => "01_PushButton"."SE01+NA0036-S1_PB", OUT_2 => "01_PushButton"."SE01+NA0037-S1_PB", OUT_3 => "01_PushButton"."SE01+NA0083-S1_PB", OUT_4 => "01_PushButton"."SE01+NA0084-S1_PB", Diag_1 =>, Diag_2 =>, Diag_3 =>, Diag_4 =>, Lamp_1 =>, Lamp_2 =>, Lamp_3 =>, Lamp_4 =>)
   END_RUNG
   // the same network as SCL:
   "n0044-ct1-el001-k30001_SN50_4"(IN_1 := "EMERGENCY PUSH BUTTON PRESSED =SE01+NA0036-S1",   // "00_Push-Button_Input"
                           IN_2 := "EMERGENCY PUSH BUTTON PRESSED =SE01+NA0037-S1",
                           IN_3 := "EMERGENCY PUSH BUTTON PRESSED =SE01+NA0083-S1",
                           IN_4 := "EMERGENCY PUSH BUTTON PRESSED =SE01+NA0084-S1",
                           ON_Tristate := "06_Settings".Tristate,
                           Bypass_ET200 := "00_Commissioning"."n0044-ct1-el001-k30001_SN50",
                           OUT_1 => "01_PushButton"."SE01+NA0036-S1_PB",
                           OUT_2 => "01_PushButton"."SE01+NA0037-S1_PB",
                           OUT_3 => "01_PushButton"."SE01+NA0083-S1_PB",
                           OUT_4 => "01_PushButton"."SE01+NA0084-S1_PB");
END_REGION

REGION Network 31: 50.045 | n0045-ct1-el002-k30001_SN50 [1]
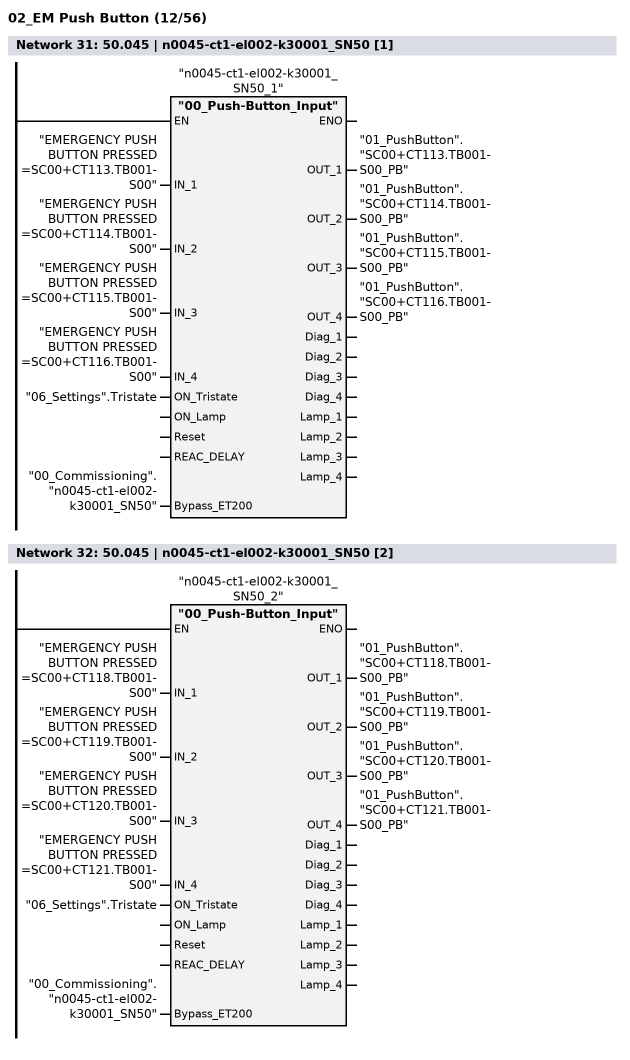
   RUNG wire#powerrail
      "n0045-ct1-el002-k30001_SN50_1"(IN_1 := "EMERGENCY PUSH BUTTON PRESSED =SC00+CT113.TB001-S00", IN_2 := "EMERGENCY PUSH BUTTON PRESSED =SC00+CT114.TB001-S00", IN_3 := "EMERGENCY PUSH BUTTON PRESSED =SC00+CT115.TB001-S00", IN_4 := "EMERGENCY PUSH BUTTON PRESSED =SC00+CT116.TB001-S00", ON_Tristate := "06_Settings".Tristate, ON_Lamp :=, Reset :=, REAC_DELAY :=, Bypass_ET200 := "00_Commissioning"."n0045-ct1-el002-k30001_SN50", OUT_1 => "01_PushButton"."SC00+CT113.TB001-S00_PB", OUT_2 => "01_PushButton"."SC00+CT114.TB001-S00_PB", OUT_3 => "01_PushButton"."SC00+CT115.TB001-S00_PB", OUT_4 => "01_PushButton"."SC00+CT116.TB001-S00_PB", Diag_1 =>, Diag_2 =>, Diag_3 =>, Diag_4 =>, Lamp_1 =>, Lamp_2 =>, Lamp_3 =>, Lamp_4 =>)
   END_RUNG
   // the same network as SCL:
   "n0045-ct1-el002-k30001_SN50_1"(IN_1 := "EMERGENCY PUSH BUTTON PRESSED =SC00+CT113.TB001-S00",   // "00_Push-Button_Input"
                           IN_2 := "EMERGENCY PUSH BUTTON PRESSED =SC00+CT114.TB001-S00",
                           IN_3 := "EMERGENCY PUSH BUTTON PRESSED =SC00+CT115.TB001-S00",
                           IN_4 := "EMERGENCY PUSH BUTTON PRESSED =SC00+CT116.TB001-S00",
                           ON_Tristate := "06_Settings".Tristate,
                           Bypass_ET200 := "00_Commissioning"."n0045-ct1-el002-k30001_SN50",
                           OUT_1 => "01_PushButton"."SC00+CT113.TB001-S00_PB",
                           OUT_2 => "01_PushButton"."SC00+CT114.TB001-S00_PB",
                           OUT_3 => "01_PushButton"."SC00+CT115.TB001-S00_PB",
                           OUT_4 => "01_PushButton"."SC00+CT116.TB001-S00_PB");
END_REGION

REGION Network 32: 50.045 | n0045-ct1-el002-k30001_SN50 [2]
   RUNG wire#powerrail
      "n0045-ct1-el002-k30001_SN50_2"(IN_1 := "EMERGENCY PUSH BUTTON PRESSED =SC00+CT118.TB001-S00", IN_2 := "EMERGENCY PUSH BUTTON PRESSED =SC00+CT119.TB001-S00", IN_3 := "EMERGENCY PUSH BUTTON PRESSED =SC00+CT120.TB001-S00", IN_4 := "EMERGENCY PUSH BUTTON PRESSED =SC00+CT121.TB001-S00", ON_Tristate := "06_Settings".Tristate, ON_Lamp :=, Reset :=, REAC_DELAY :=, Bypass_ET200 := "00_Commissioning"."n0045-ct1-el002-k30001_SN50", OUT_1 => "01_PushButton"."SC00+CT118.TB001-S00_PB", OUT_2 => "01_PushButton"."SC00+CT119.TB001-S00_PB", OUT_3 => "01_PushButton"."SC00+CT120.TB001-S00_PB", OUT_4 => "01_PushButton"."SC00+CT121.TB001-S00_PB", Diag_1 =>, Diag_2 =>, Diag_3 =>, Diag_4 =>, Lamp_1 =>, Lamp_2 =>, Lamp_3 =>, Lamp_4 =>)
   END_RUNG
   // the same network as SCL:
   "n0045-ct1-el002-k30001_SN50_2"(IN_1 := "EMERGENCY PUSH BUTTON PRESSED =SC00+CT118.TB001-S00",   // "00_Push-Button_Input"
                           IN_2 := "EMERGENCY PUSH BUTTON PRESSED =SC00+CT119.TB001-S00",
                           IN_3 := "EMERGENCY PUSH BUTTON PRESSED =SC00+CT120.TB001-S00",
                           IN_4 := "EMERGENCY PUSH BUTTON PRESSED =SC00+CT121.TB001-S00",
                           ON_Tristate := "06_Settings".Tristate,
                           Bypass_ET200 := "00_Commissioning"."n0045-ct1-el002-k30001_SN50",
                           OUT_1 => "01_PushButton"."SC00+CT118.TB001-S00_PB",
                           OUT_2 => "01_PushButton"."SC00+CT119.TB001-S00_PB",
                           OUT_3 => "01_PushButton"."SC00+CT120.TB001-S00_PB",
                           OUT_4 => "01_PushButton"."SC00+CT121.TB001-S00_PB");
END_REGION

REGION Network 33: 50.045 | n0045-ct1-el002-k30001_SN50 [3]
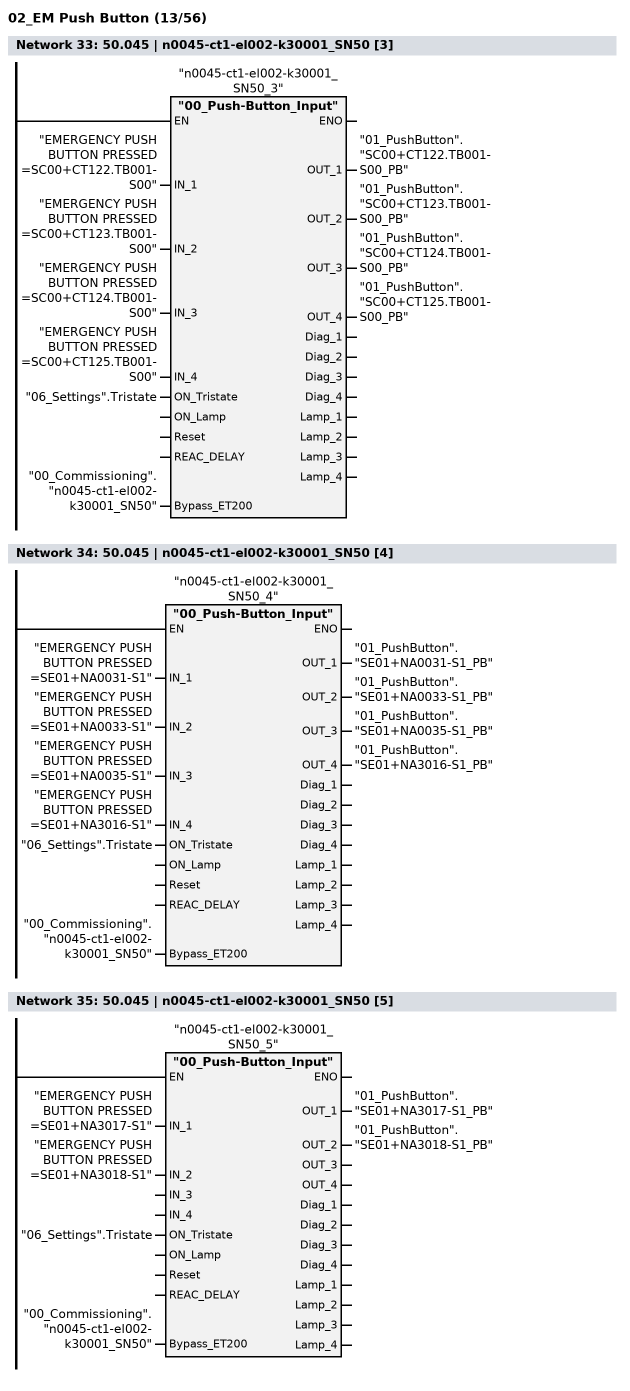
   RUNG wire#powerrail
      "n0045-ct1-el002-k30001_SN50_3"(IN_1 := "EMERGENCY PUSH BUTTON PRESSED =SC00+CT122.TB001-S00", IN_2 := "EMERGENCY PUSH BUTTON PRESSED =SC00+CT123.TB001-S00", IN_3 := "EMERGENCY PUSH BUTTON PRESSED =SC00+CT124.TB001-S00", IN_4 := "EMERGENCY PUSH BUTTON PRESSED =SC00+CT125.TB001-S00", ON_Tristate := "06_Settings".Tristate, ON_Lamp :=, Reset :=, REAC_DELAY :=, Bypass_ET200 := "00_Commissioning"."n0045-ct1-el002-k30001_SN50", OUT_1 => "01_PushButton"."SC00+CT122.TB001-S00_PB", OUT_2 => "01_PushButton"."SC00+CT123.TB001-S00_PB", OUT_3 => "01_PushButton"."SC00+CT124.TB001-S00_PB", OUT_4 => "01_PushButton"."SC00+CT125.TB001-S00_PB", Diag_1 =>, Diag_2 =>, Diag_3 =>, Diag_4 =>, Lamp_1 =>, Lamp_2 =>, Lamp_3 =>, Lamp_4 =>)
   END_RUNG
   // the same network as SCL:
   "n0045-ct1-el002-k30001_SN50_3"(IN_1 := "EMERGENCY PUSH BUTTON PRESSED =SC00+CT122.TB001-S00",   // "00_Push-Button_Input"
                           IN_2 := "EMERGENCY PUSH BUTTON PRESSED =SC00+CT123.TB001-S00",
                           IN_3 := "EMERGENCY PUSH BUTTON PRESSED =SC00+CT124.TB001-S00",
                           IN_4 := "EMERGENCY PUSH BUTTON PRESSED =SC00+CT125.TB001-S00",
                           ON_Tristate := "06_Settings".Tristate,
                           Bypass_ET200 := "00_Commissioning"."n0045-ct1-el002-k30001_SN50",
                           OUT_1 => "01_PushButton"."SC00+CT122.TB001-S00_PB",
                           OUT_2 => "01_PushButton"."SC00+CT123.TB001-S00_PB",
                           OUT_3 => "01_PushButton"."SC00+CT124.TB001-S00_PB",
                           OUT_4 => "01_PushButton"."SC00+CT125.TB001-S00_PB");
END_REGION

REGION Network 34: 50.045 | n0045-ct1-el002-k30001_SN50 [4]
   RUNG wire#powerrail
      "n0045-ct1-el002-k30001_SN50_4"(IN_1 := "EMERGENCY PUSH BUTTON PRESSED =SE01+NA0031-S1", IN_2 := "EMERGENCY PUSH BUTTON PRESSED =SE01+NA0033-S1", IN_3 := "EMERGENCY PUSH BUTTON PRESSED =SE01+NA0035-S1", IN_4 := "EMERGENCY PUSH BUTTON PRESSED =SE01+NA3016-S1", ON_Tristate := "06_Settings".Tristate, ON_Lamp :=, Reset :=, REAC_DELAY :=, Bypass_ET200 := "00_Commissioning"."n0045-ct1-el002-k30001_SN50", OUT_1 => "01_PushButton"."SE01+NA0031-S1_PB", OUT_2 => "01_PushButton"."SE01+NA0033-S1_PB", OUT_3 => "01_PushButton"."SE01+NA0035-S1_PB", OUT_4 => "01_PushButton"."SE01+NA3016-S1_PB", Diag_1 =>, Diag_2 =>, Diag_3 =>, Diag_4 =>, Lamp_1 =>, Lamp_2 =>, Lamp_3 =>, Lamp_4 =>)
   END_RUNG
   // the same network as SCL:
   "n0045-ct1-el002-k30001_SN50_4"(IN_1 := "EMERGENCY PUSH BUTTON PRESSED =SE01+NA0031-S1",   // "00_Push-Button_Input"
                           IN_2 := "EMERGENCY PUSH BUTTON PRESSED =SE01+NA0033-S1",
                           IN_3 := "EMERGENCY PUSH BUTTON PRESSED =SE01+NA0035-S1",
                           IN_4 := "EMERGENCY PUSH BUTTON PRESSED =SE01+NA3016-S1",
                           ON_Tristate := "06_Settings".Tristate,
                           Bypass_ET200 := "00_Commissioning"."n0045-ct1-el002-k30001_SN50",
                           OUT_1 => "01_PushButton"."SE01+NA0031-S1_PB",
                           OUT_2 => "01_PushButton"."SE01+NA0033-S1_PB",
                           OUT_3 => "01_PushButton"."SE01+NA0035-S1_PB",
                           OUT_4 => "01_PushButton"."SE01+NA3016-S1_PB");
END_REGION

REGION Network 35: 50.045 | n0045-ct1-el002-k30001_SN50 [5]
   RUNG wire#powerrail
      "n0045-ct1-el002-k30001_SN50_5"(IN_1 := "EMERGENCY PUSH BUTTON PRESSED =SE01+NA3017-S1", IN_2 := "EMERGENCY PUSH BUTTON PRESSED =SE01+NA3018-S1", IN_3 :=, IN_4 :=, ON_Tristate := "06_Settings".Tristate, ON_Lamp :=, Reset :=, REAC_DELAY :=, Bypass_ET200 := "00_Commissioning"."n0045-ct1-el002-k30001_SN50", OUT_1 => "01_PushButton"."SE01+NA3017-S1_PB", OUT_2 => "01_PushButton"."SE01+NA3018-S1_PB", OUT_3 =>, OUT_4 =>, Diag_1 =>, Diag_2 =>, Diag_3 =>, Diag_4 =>, Lamp_1 =>, Lamp_2 =>, Lamp_3 =>, Lamp_4 =>)
   END_RUNG
   // the same network as SCL:
   "n0045-ct1-el002-k30001_SN50_5"(IN_1 := "EMERGENCY PUSH BUTTON PRESSED =SE01+NA3017-S1",   // "00_Push-Button_Input"
                           IN_2 := "EMERGENCY PUSH BUTTON PRESSED =SE01+NA3018-S1",
                           ON_Tristate := "06_Settings".Tristate,
                           Bypass_ET200 := "00_Commissioning"."n0045-ct1-el002-k30001_SN50",
                           OUT_1 => "01_PushButton"."SE01+NA3017-S1_PB",
                           OUT_2 => "01_PushButton"."SE01+NA3018-S1_PB");
END_REGION

REGION Network 36: 50.046 | n0046-ct1-el003-k30001_SN50 [1]
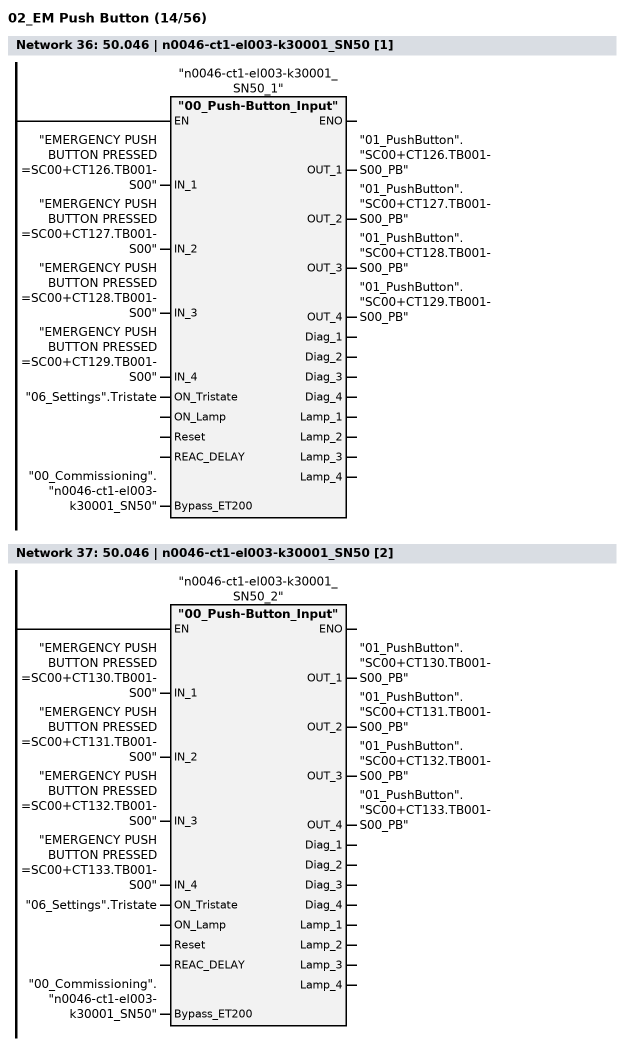
   RUNG wire#powerrail
      "n0046-ct1-el003-k30001_SN50_1"(IN_1 := "EMERGENCY PUSH BUTTON PRESSED =SC00+CT126.TB001-S00", IN_2 := "EMERGENCY PUSH BUTTON PRESSED =SC00+CT127.TB001-S00", IN_3 := "EMERGENCY PUSH BUTTON PRESSED =SC00+CT128.TB001-S00", IN_4 := "EMERGENCY PUSH BUTTON PRESSED =SC00+CT129.TB001-S00", ON_Tristate := "06_Settings".Tristate, ON_Lamp :=, Reset :=, REAC_DELAY :=, Bypass_ET200 := "00_Commissioning"."n0046-ct1-el003-k30001_SN50", OUT_1 => "01_PushButton"."SC00+CT126.TB001-S00_PB", OUT_2 => "01_PushButton"."SC00+CT127.TB001-S00_PB", OUT_3 => "01_PushButton"."SC00+CT128.TB001-S00_PB", OUT_4 => "01_PushButton"."SC00+CT129.TB001-S00_PB", Diag_1 =>, Diag_2 =>, Diag_3 =>, Diag_4 =>, Lamp_1 =>, Lamp_2 =>, Lamp_3 =>, Lamp_4 =>)
   END_RUNG
   // the same network as SCL:
   "n0046-ct1-el003-k30001_SN50_1"(IN_1 := "EMERGENCY PUSH BUTTON PRESSED =SC00+CT126.TB001-S00",   // "00_Push-Button_Input"
                           IN_2 := "EMERGENCY PUSH BUTTON PRESSED =SC00+CT127.TB001-S00",
                           IN_3 := "EMERGENCY PUSH BUTTON PRESSED =SC00+CT128.TB001-S00",
                           IN_4 := "EMERGENCY PUSH BUTTON PRESSED =SC00+CT129.TB001-S00",
                           ON_Tristate := "06_Settings".Tristate,
                           Bypass_ET200 := "00_Commissioning"."n0046-ct1-el003-k30001_SN50",
                           OUT_1 => "01_PushButton"."SC00+CT126.TB001-S00_PB",
                           OUT_2 => "01_PushButton"."SC00+CT127.TB001-S00_PB",
                           OUT_3 => "01_PushButton"."SC00+CT128.TB001-S00_PB",
                           OUT_4 => "01_PushButton"."SC00+CT129.TB001-S00_PB");
END_REGION

REGION Network 37: 50.046 | n0046-ct1-el003-k30001_SN50 [2]
   RUNG wire#powerrail
      "n0046-ct1-el003-k30001_SN50_2"(IN_1 := "EMERGENCY PUSH BUTTON PRESSED =SC00+CT130.TB001-S00", IN_2 := "EMERGENCY PUSH BUTTON PRESSED =SC00+CT131.TB001-S00", IN_3 := "EMERGENCY PUSH BUTTON PRESSED =SC00+CT132.TB001-S00", IN_4 := "EMERGENCY PUSH BUTTON PRESSED =SC00+CT133.TB001-S00", ON_Tristate := "06_Settings".Tristate, ON_Lamp :=, Reset :=, REAC_DELAY :=, Bypass_ET200 := "00_Commissioning"."n0046-ct1-el003-k30001_SN50", OUT_1 => "01_PushButton"."SC00+CT130.TB001-S00_PB", OUT_2 => "01_PushButton"."SC00+CT131.TB001-S00_PB", OUT_3 => "01_PushButton"."SC00+CT132.TB001-S00_PB", OUT_4 => "01_PushButton"."SC00+CT133.TB001-S00_PB", Diag_1 =>, Diag_2 =>, Diag_3 =>, Diag_4 =>, Lamp_1 =>, Lamp_2 =>, Lamp_3 =>, Lamp_4 =>)
   END_RUNG
   // the same network as SCL:
   "n0046-ct1-el003-k30001_SN50_2"(IN_1 := "EMERGENCY PUSH BUTTON PRESSED =SC00+CT130.TB001-S00",   // "00_Push-Button_Input"
                           IN_2 := "EMERGENCY PUSH BUTTON PRESSED =SC00+CT131.TB001-S00",
                           IN_3 := "EMERGENCY PUSH BUTTON PRESSED =SC00+CT132.TB001-S00",
                           IN_4 := "EMERGENCY PUSH BUTTON PRESSED =SC00+CT133.TB001-S00",
                           ON_Tristate := "06_Settings".Tristate,
                           Bypass_ET200 := "00_Commissioning"."n0046-ct1-el003-k30001_SN50",
                           OUT_1 => "01_PushButton"."SC00+CT130.TB001-S00_PB",
                           OUT_2 => "01_PushButton"."SC00+CT131.TB001-S00_PB",
                           OUT_3 => "01_PushButton"."SC00+CT132.TB001-S00_PB",
                           OUT_4 => "01_PushButton"."SC00+CT133.TB001-S00_PB");
END_REGION

REGION Network 38: 50.046 | n0046-ct1-el003-k30001_SN50 [3]
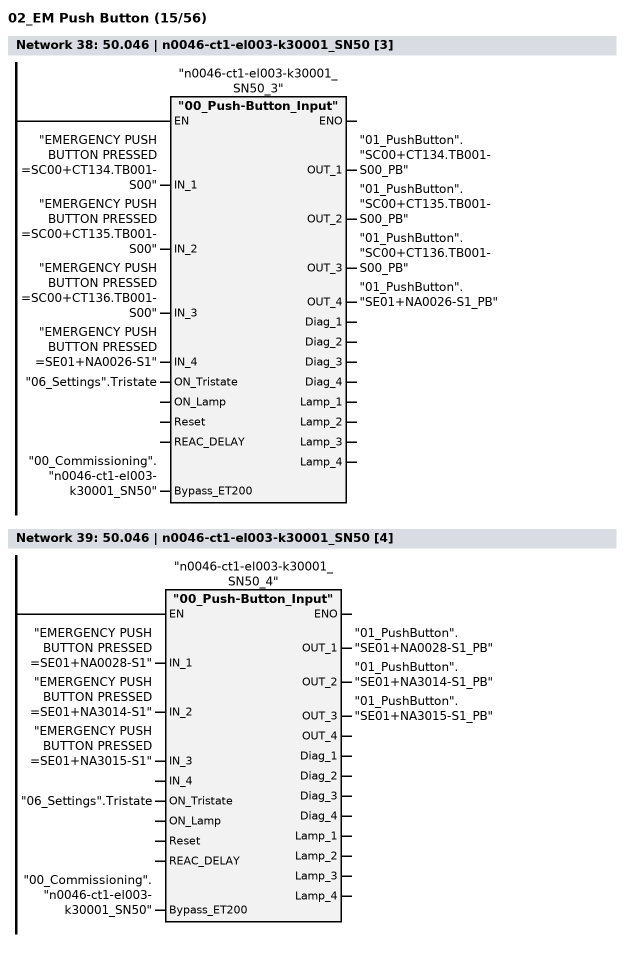
   RUNG wire#powerrail
      "n0046-ct1-el003-k30001_SN50_3"(IN_1 := "EMERGENCY PUSH BUTTON PRESSED =SC00+CT134.TB001-S00", IN_2 := "EMERGENCY PUSH BUTTON PRESSED =SC00+CT135.TB001-S00", IN_3 := "EMERGENCY PUSH BUTTON PRESSED =SC00+CT136.TB001-S00", IN_4 := "EMERGENCY PUSH BUTTON PRESSED =SE01+NA0026-S1", ON_Tristate := "06_Settings".Tristate, ON_Lamp :=, Reset :=, REAC_DELAY :=, Bypass_ET200 := "00_Commissioning"."n0046-ct1-el003-k30001_SN50", OUT_1 => "01_PushButton"."SC00+CT134.TB001-S00_PB", OUT_2 => "01_PushButton"."SC00+CT135.TB001-S00_PB", OUT_3 => "01_PushButton"."SC00+CT136.TB001-S00_PB", OUT_4 => "01_PushButton"."SE01+NA0026-S1_PB", Diag_1 =>, Diag_2 =>, Diag_3 =>, Diag_4 =>, Lamp_1 =>, Lamp_2 =>, Lamp_3 =>, Lamp_4 =>)
   END_RUNG
   // the same network as SCL:
   "n0046-ct1-el003-k30001_SN50_3"(IN_1 := "EMERGENCY PUSH BUTTON PRESSED =SC00+CT134.TB001-S00",   // "00_Push-Button_Input"
                           IN_2 := "EMERGENCY PUSH BUTTON PRESSED =SC00+CT135.TB001-S00",
                           IN_3 := "EMERGENCY PUSH BUTTON PRESSED =SC00+CT136.TB001-S00",
                           IN_4 := "EMERGENCY PUSH BUTTON PRESSED =SE01+NA0026-S1",
                           ON_Tristate := "06_Settings".Tristate,
                           Bypass_ET200 := "00_Commissioning"."n0046-ct1-el003-k30001_SN50",
                           OUT_1 => "01_PushButton"."SC00+CT134.TB001-S00_PB",
                           OUT_2 => "01_PushButton"."SC00+CT135.TB001-S00_PB",
                           OUT_3 => "01_PushButton"."SC00+CT136.TB001-S00_PB",
                           OUT_4 => "01_PushButton"."SE01+NA0026-S1_PB");
END_REGION

REGION Network 39: 50.046 | n0046-ct1-el003-k30001_SN50 [4]
   RUNG wire#powerrail
      "n0046-ct1-el003-k30001_SN50_4"(IN_1 := "EMERGENCY PUSH BUTTON PRESSED =SE01+NA0028-S1", IN_2 := "EMERGENCY PUSH BUTTON PRESSED =SE01+NA3014-S1", IN_3 := "EMERGENCY PUSH BUTTON PRESSED =SE01+NA3015-S1", IN_4 :=, ON_Tristate := "06_Settings".Tristate, ON_Lamp :=, Reset :=, REAC_DELAY :=, Bypass_ET200 := "00_Commissioning"."n0046-ct1-el003-k30001_SN50", OUT_1 => "01_PushButton"."SE01+NA0028-S1_PB", OUT_2 => "01_PushButton"."SE01+NA3014-S1_PB", OUT_3 => "01_PushButton"."SE01+NA3015-S1_PB", OUT_4 =>, Diag_1 =>, Diag_2 =>, Diag_3 =>, Diag_4 =>, Lamp_1 =>, Lamp_2 =>, Lamp_3 =>, Lamp_4 =>)
   END_RUNG
   // the same network as SCL:
   "n0046-ct1-el003-k30001_SN50_4"(IN_1 := "EMERGENCY PUSH BUTTON PRESSED =SE01+NA0028-S1",   // "00_Push-Button_Input"
                           IN_2 := "EMERGENCY PUSH BUTTON PRESSED =SE01+NA3014-S1",
                           IN_3 := "EMERGENCY PUSH BUTTON PRESSED =SE01+NA3015-S1",
                           ON_Tristate := "06_Settings".Tristate,
                           Bypass_ET200 := "00_Commissioning"."n0046-ct1-el003-k30001_SN50",
                           OUT_1 => "01_PushButton"."SE01+NA0028-S1_PB",
                           OUT_2 => "01_PushButton"."SE01+NA3014-S1_PB",
                           OUT_3 => "01_PushButton"."SE01+NA3015-S1_PB");
END_REGION

REGION Network 40: 50.050 | n0050-uc13-el001-k30001_SN50 [1]
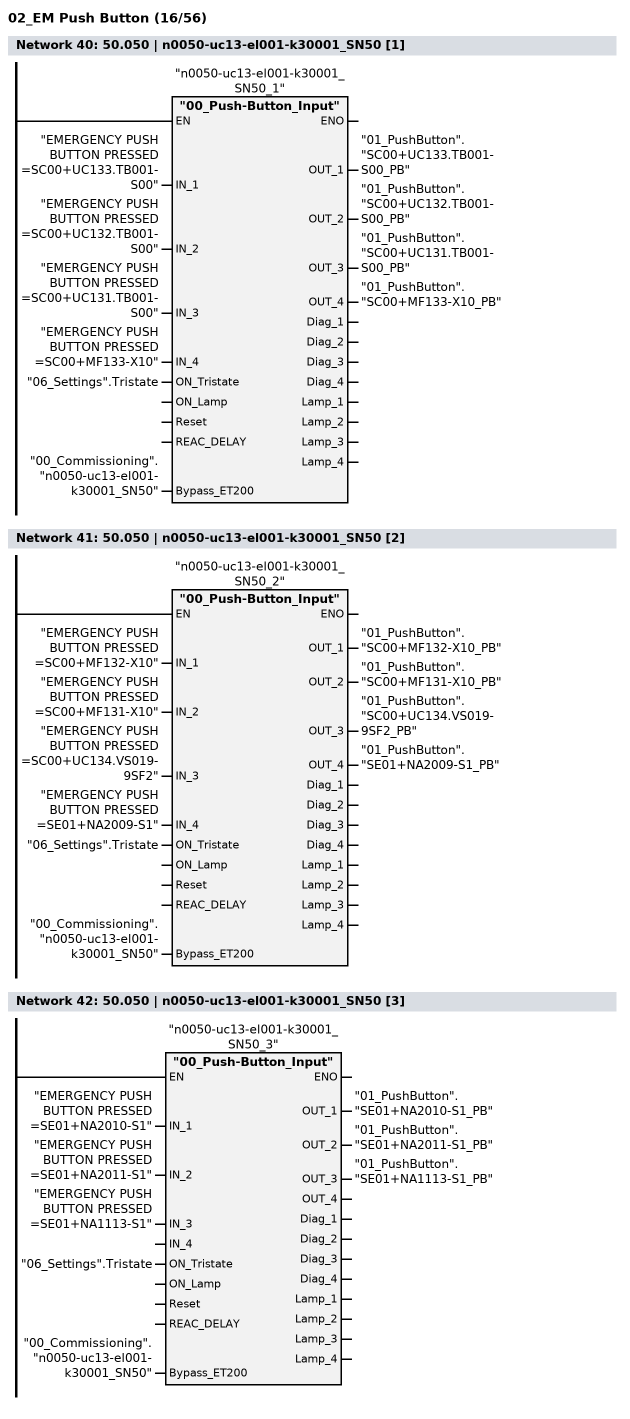
   RUNG wire#powerrail
      "n0050-uc13-el001-k30001_SN50_1"(IN_1 := "EMERGENCY PUSH BUTTON PRESSED =SC00+UC133.TB001-S00", IN_2 := "EMERGENCY PUSH BUTTON PRESSED =SC00+UC132.TB001-S00", IN_3 := "EMERGENCY PUSH BUTTON PRESSED =SC00+UC131.TB001-S00", IN_4 := "EMERGENCY PUSH BUTTON PRESSED =SC00+MF133-X10", ON_Tristate := "06_Settings".Tristate, ON_Lamp :=, Reset :=, REAC_DELAY :=, Bypass_ET200 := "00_Commissioning"."n0050-uc13-el001-k30001_SN50", OUT_1 => "01_PushButton"."SC00+UC133.TB001-S00_PB", OUT_2 => "01_PushButton"."SC00+UC132.TB001-S00_PB", OUT_3 => "01_PushButton"."SC00+UC131.TB001-S00_PB", OUT_4 => "01_PushButton"."SC00+MF133-X10_PB", Diag_1 =>, Diag_2 =>, Diag_3 =>, Diag_4 =>, Lamp_1 =>, Lamp_2 =>, Lamp_3 =>, Lamp_4 =>)
   END_RUNG
   // the same network as SCL:
   "n0050-uc13-el001-k30001_SN50_1"(IN_1 := "EMERGENCY PUSH BUTTON PRESSED =SC00+UC133.TB001-S00",   // "00_Push-Button_Input"
                           IN_2 := "EMERGENCY PUSH BUTTON PRESSED =SC00+UC132.TB001-S00",
                           IN_3 := "EMERGENCY PUSH BUTTON PRESSED =SC00+UC131.TB001-S00",
                           IN_4 := "EMERGENCY PUSH BUTTON PRESSED =SC00+MF133-X10",
                           ON_Tristate := "06_Settings".Tristate,
                           Bypass_ET200 := "00_Commissioning"."n0050-uc13-el001-k30001_SN50",
                           OUT_1 => "01_PushButton"."SC00+UC133.TB001-S00_PB",
                           OUT_2 => "01_PushButton"."SC00+UC132.TB001-S00_PB",
                           OUT_3 => "01_PushButton"."SC00+UC131.TB001-S00_PB",
                           OUT_4 => "01_PushButton"."SC00+MF133-X10_PB");
END_REGION

REGION Network 41: 50.050 | n0050-uc13-el001-k30001_SN50 [2]
   RUNG wire#powerrail
      "n0050-uc13-el001-k30001_SN50_2"(IN_1 := "EMERGENCY PUSH BUTTON PRESSED =SC00+MF132-X10", IN_2 := "EMERGENCY PUSH BUTTON PRESSED =SC00+MF131-X10", IN_3 := "EMERGENCY PUSH BUTTON PRESSED =SC00+UC134.VS019-9SF2", IN_4 := "EMERGENCY PUSH BUTTON PRESSED =SE01+NA2009-S1", ON_Tristate := "06_Settings".Tristate, ON_Lamp :=, Reset :=, REAC_DELAY :=, Bypass_ET200 := "00_Commissioning"."n0050-uc13-el001-k30001_SN50", OUT_1 => "01_PushButton"."SC00+MF132-X10_PB", OUT_2 => "01_PushButton"."SC00+MF131-X10_PB", OUT_3 => "01_PushButton"."SC00+UC134.VS019-9SF2_PB", OUT_4 => "01_PushButton"."SE01+NA2009-S1_PB", Diag_1 =>, Diag_2 =>, Diag_3 =>, Diag_4 =>, Lamp_1 =>, Lamp_2 =>, Lamp_3 =>, Lamp_4 =>)
   END_RUNG
   // the same network as SCL:
   "n0050-uc13-el001-k30001_SN50_2"(IN_1 := "EMERGENCY PUSH BUTTON PRESSED =SC00+MF132-X10",   // "00_Push-Button_Input"
                           IN_2 := "EMERGENCY PUSH BUTTON PRESSED =SC00+MF131-X10",
                           IN_3 := "EMERGENCY PUSH BUTTON PRESSED =SC00+UC134.VS019-9SF2",
                           IN_4 := "EMERGENCY PUSH BUTTON PRESSED =SE01+NA2009-S1",
                           ON_Tristate := "06_Settings".Tristate,
                           Bypass_ET200 := "00_Commissioning"."n0050-uc13-el001-k30001_SN50",
                           OUT_1 => "01_PushButton"."SC00+MF132-X10_PB",
                           OUT_2 => "01_PushButton"."SC00+MF131-X10_PB",
                           OUT_3 => "01_PushButton"."SC00+UC134.VS019-9SF2_PB",
                           OUT_4 => "01_PushButton"."SE01+NA2009-S1_PB");
END_REGION

REGION Network 42: 50.050 | n0050-uc13-el001-k30001_SN50 [3]
   RUNG wire#powerrail
      "n0050-uc13-el001-k30001_SN50_3"(IN_1 := "EMERGENCY PUSH BUTTON PRESSED =SE01+NA2010-S1", IN_2 := "EMERGENCY PUSH BUTTON PRESSED =SE01+NA2011-S1", IN_3 := "EMERGENCY PUSH BUTTON PRESSED =SE01+NA1113-S1", IN_4 :=, ON_Tristate := "06_Settings".Tristate, ON_Lamp :=, Reset :=, REAC_DELAY :=, Bypass_ET200 := "00_Commissioning"."n0050-uc13-el001-k30001_SN50", OUT_1 => "01_PushButton"."SE01+NA2010-S1_PB", OUT_2 => "01_PushButton"."SE01+NA2011-S1_PB", OUT_3 => "01_PushButton"."SE01+NA1113-S1_PB", OUT_4 =>, Diag_1 =>, Diag_2 =>, Diag_3 =>, Diag_4 =>, Lamp_1 =>, Lamp_2 =>, Lamp_3 =>, Lamp_4 =>)
   END_RUNG
   // the same network as SCL:
   "n0050-uc13-el001-k30001_SN50_3"(IN_1 := "EMERGENCY PUSH BUTTON PRESSED =SE01+NA2010-S1",   // "00_Push-Button_Input"
                           IN_2 := "EMERGENCY PUSH BUTTON PRESSED =SE01+NA2011-S1",
                           IN_3 := "EMERGENCY PUSH BUTTON PRESSED =SE01+NA1113-S1",
                           ON_Tristate := "06_Settings".Tristate,
                           Bypass_ET200 := "00_Commissioning"."n0050-uc13-el001-k30001_SN50",
                           OUT_1 => "01_PushButton"."SE01+NA2010-S1_PB",
                           OUT_2 => "01_PushButton"."SE01+NA2011-S1_PB",
                           OUT_3 => "01_PushButton"."SE01+NA1113-S1_PB");
END_REGION

REGION Network 43: 50.051 | n0051-uc134-xn10_SN50 [1]
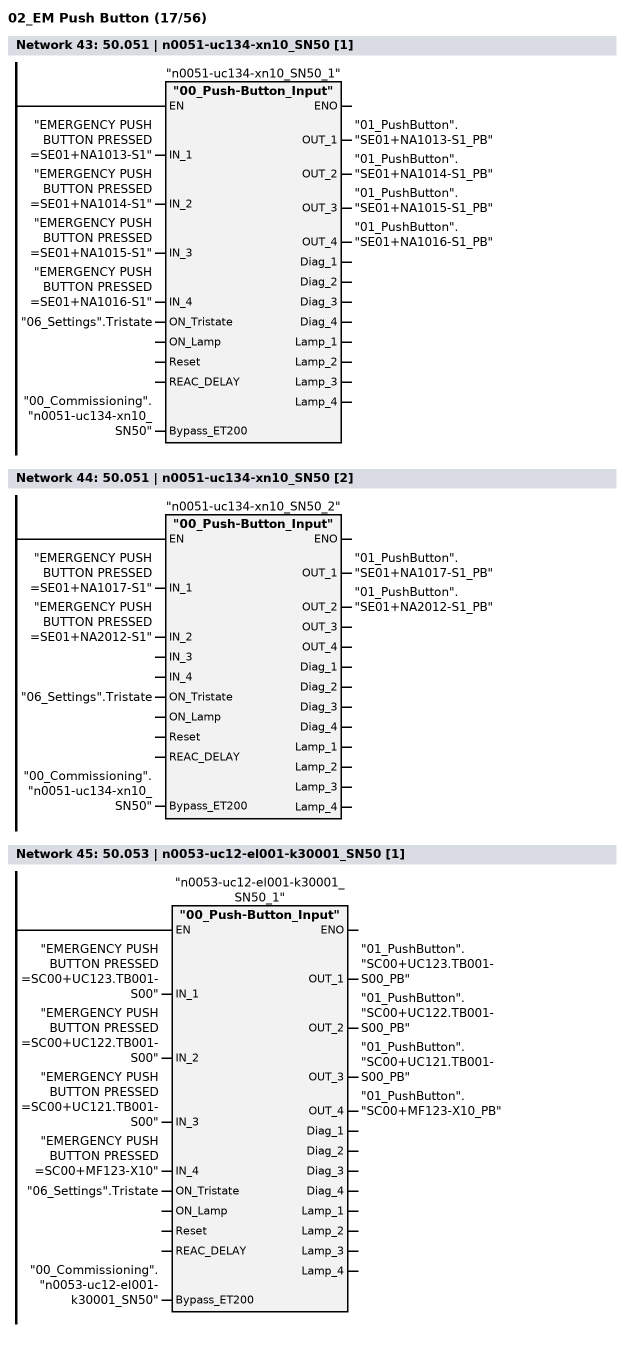
   RUNG wire#powerrail
      "n0051-uc134-xn10_SN50_1"(IN_1 := "EMERGENCY PUSH BUTTON PRESSED =SE01+NA1013-S1", IN_2 := "EMERGENCY PUSH BUTTON PRESSED =SE01+NA1014-S1", IN_3 := "EMERGENCY PUSH BUTTON PRESSED =SE01+NA1015-S1", IN_4 := "EMERGENCY PUSH BUTTON PRESSED =SE01+NA1016-S1", ON_Tristate := "06_Settings".Tristate, ON_Lamp :=, Reset :=, REAC_DELAY :=, Bypass_ET200 := "00_Commissioning"."n0051-uc134-xn10_SN50", OUT_1 => "01_PushButton"."SE01+NA1013-S1_PB", OUT_2 => "01_PushButton"."SE01+NA1014-S1_PB", OUT_3 => "01_PushButton"."SE01+NA1015-S1_PB", OUT_4 => "01_PushButton"."SE01+NA1016-S1_PB", Diag_1 =>, Diag_2 =>, Diag_3 =>, Diag_4 =>, Lamp_1 =>, Lamp_2 =>, Lamp_3 =>, Lamp_4 =>)
   END_RUNG
   // the same network as SCL:
   "n0051-uc134-xn10_SN50_1"(IN_1 := "EMERGENCY PUSH BUTTON PRESSED =SE01+NA1013-S1",   // "00_Push-Button_Input"
                           IN_2 := "EMERGENCY PUSH BUTTON PRESSED =SE01+NA1014-S1",
                           IN_3 := "EMERGENCY PUSH BUTTON PRESSED =SE01+NA1015-S1",
                           IN_4 := "EMERGENCY PUSH BUTTON PRESSED =SE01+NA1016-S1",
                           ON_Tristate := "06_Settings".Tristate,
                           Bypass_ET200 := "00_Commissioning"."n0051-uc134-xn10_SN50",
                           OUT_1 => "01_PushButton"."SE01+NA1013-S1_PB",
                           OUT_2 => "01_PushButton"."SE01+NA1014-S1_PB",
                           OUT_3 => "01_PushButton"."SE01+NA1015-S1_PB",
                           OUT_4 => "01_PushButton"."SE01+NA1016-S1_PB");
END_REGION

REGION Network 44: 50.051 | n0051-uc134-xn10_SN50 [2]
   RUNG wire#powerrail
      "n0051-uc134-xn10_SN50_2"(IN_1 := "EMERGENCY PUSH BUTTON PRESSED =SE01+NA1017-S1", IN_2 := "EMERGENCY PUSH BUTTON PRESSED =SE01+NA2012-S1", IN_3 :=, IN_4 :=, ON_Tristate := "06_Settings".Tristate, ON_Lamp :=, Reset :=, REAC_DELAY :=, Bypass_ET200 := "00_Commissioning"."n0051-uc134-xn10_SN50", OUT_1 => "01_PushButton"."SE01+NA1017-S1_PB", OUT_2 => "01_PushButton"."SE01+NA2012-S1_PB", OUT_3 =>, OUT_4 =>, Diag_1 =>, Diag_2 =>, Diag_3 =>, Diag_4 =>, Lamp_1 =>, Lamp_2 =>, Lamp_3 =>, Lamp_4 =>)
   END_RUNG
   // the same network as SCL:
   "n0051-uc134-xn10_SN50_2"(IN_1 := "EMERGENCY PUSH BUTTON PRESSED =SE01+NA1017-S1",   // "00_Push-Button_Input"
                           IN_2 := "EMERGENCY PUSH BUTTON PRESSED =SE01+NA2012-S1",
                           ON_Tristate := "06_Settings".Tristate,
                           Bypass_ET200 := "00_Commissioning"."n0051-uc134-xn10_SN50",
                           OUT_1 => "01_PushButton"."SE01+NA1017-S1_PB",
                           OUT_2 => "01_PushButton"."SE01+NA2012-S1_PB");
END_REGION

REGION Network 45: 50.053 | n0053-uc12-el001-k30001_SN50 [1]
   RUNG wire#powerrail
      "n0053-uc12-el001-k30001_SN50_1"(IN_1 := "EMERGENCY PUSH BUTTON PRESSED =SC00+UC123.TB001-S00", IN_2 := "EMERGENCY PUSH BUTTON PRESSED =SC00+UC122.TB001-S00", IN_3 := "EMERGENCY PUSH BUTTON PRESSED =SC00+UC121.TB001-S00", IN_4 := "EMERGENCY PUSH BUTTON PRESSED =SC00+MF123-X10", ON_Tristate := "06_Settings".Tristate, ON_Lamp :=, Reset :=, REAC_DELAY :=, Bypass_ET200 := "00_Commissioning"."n0053-uc12-el001-k30001_SN50", OUT_1 => "01_PushButton"."SC00+UC123.TB001-S00_PB", OUT_2 => "01_PushButton"."SC00+UC122.TB001-S00_PB", OUT_3 => "01_PushButton"."SC00+UC121.TB001-S00_PB", OUT_4 => "01_PushButton"."SC00+MF123-X10_PB", Diag_1 =>, Diag_2 =>, Diag_3 =>, Diag_4 =>, Lamp_1 =>, Lamp_2 =>, Lamp_3 =>, Lamp_4 =>)
   END_RUNG
   // the same network as SCL:
   "n0053-uc12-el001-k30001_SN50_1"(IN_1 := "EMERGENCY PUSH BUTTON PRESSED =SC00+UC123.TB001-S00",   // "00_Push-Button_Input"
                           IN_2 := "EMERGENCY PUSH BUTTON PRESSED =SC00+UC122.TB001-S00",
                           IN_3 := "EMERGENCY PUSH BUTTON PRESSED =SC00+UC121.TB001-S00",
                           IN_4 := "EMERGENCY PUSH BUTTON PRESSED =SC00+MF123-X10",
                           ON_Tristate := "06_Settings".Tristate,
                           Bypass_ET200 := "00_Commissioning"."n0053-uc12-el001-k30001_SN50",
                           OUT_1 => "01_PushButton"."SC00+UC123.TB001-S00_PB",
                           OUT_2 => "01_PushButton"."SC00+UC122.TB001-S00_PB",
                           OUT_3 => "01_PushButton"."SC00+UC121.TB001-S00_PB",
                           OUT_4 => "01_PushButton"."SC00+MF123-X10_PB");
END_REGION

REGION Network 46: 50.053 | n0053-uc12-el001-k30001_SN50 [2]
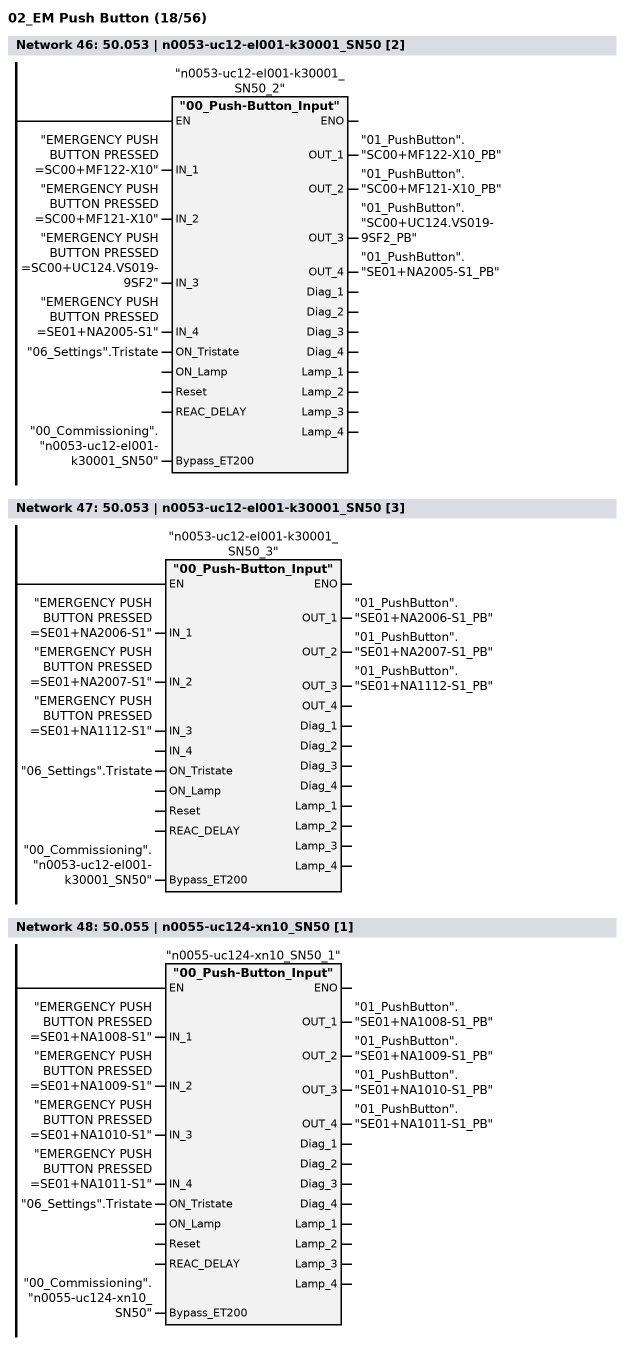
   RUNG wire#powerrail
      "n0053-uc12-el001-k30001_SN50_2"(IN_1 := "EMERGENCY PUSH BUTTON PRESSED =SC00+MF122-X10", IN_2 := "EMERGENCY PUSH BUTTON PRESSED =SC00+MF121-X10", IN_3 := "EMERGENCY PUSH BUTTON PRESSED =SC00+UC124.VS019-9SF2", IN_4 := "EMERGENCY PUSH BUTTON PRESSED =SE01+NA2005-S1", ON_Tristate := "06_Settings".Tristate, ON_Lamp :=, Reset :=, REAC_DELAY :=, Bypass_ET200 := "00_Commissioning"."n0053-uc12-el001-k30001_SN50", OUT_1 => "01_PushButton"."SC00+MF122-X10_PB", OUT_2 => "01_PushButton"."SC00+MF121-X10_PB", OUT_3 => "01_PushButton"."SC00+UC124.VS019-9SF2_PB", OUT_4 => "01_PushButton"."SE01+NA2005-S1_PB", Diag_1 =>, Diag_2 =>, Diag_3 =>, Diag_4 =>, Lamp_1 =>, Lamp_2 =>, Lamp_3 =>, Lamp_4 =>)
   END_RUNG
   // the same network as SCL:
   "n0053-uc12-el001-k30001_SN50_2"(IN_1 := "EMERGENCY PUSH BUTTON PRESSED =SC00+MF122-X10",   // "00_Push-Button_Input"
                           IN_2 := "EMERGENCY PUSH BUTTON PRESSED =SC00+MF121-X10",
                           IN_3 := "EMERGENCY PUSH BUTTON PRESSED =SC00+UC124.VS019-9SF2",
                           IN_4 := "EMERGENCY PUSH BUTTON PRESSED =SE01+NA2005-S1",
                           ON_Tristate := "06_Settings".Tristate,
                           Bypass_ET200 := "00_Commissioning"."n0053-uc12-el001-k30001_SN50",
                           OUT_1 => "01_PushButton"."SC00+MF122-X10_PB",
                           OUT_2 => "01_PushButton"."SC00+MF121-X10_PB",
                           OUT_3 => "01_PushButton"."SC00+UC124.VS019-9SF2_PB",
                           OUT_4 => "01_PushButton"."SE01+NA2005-S1_PB");
END_REGION

REGION Network 47: 50.053 | n0053-uc12-el001-k30001_SN50 [3]
   RUNG wire#powerrail
      "n0053-uc12-el001-k30001_SN50_3"(IN_1 := "EMERGENCY PUSH BUTTON PRESSED =SE01+NA2006-S1", IN_2 := "EMERGENCY PUSH BUTTON PRESSED =SE01+NA2007-S1", IN_3 := "EMERGENCY PUSH BUTTON PRESSED =SE01+NA1112-S1", IN_4 :=, ON_Tristate := "06_Settings".Tristate, ON_Lamp :=, Reset :=, REAC_DELAY :=, Bypass_ET200 := "00_Commissioning"."n0053-uc12-el001-k30001_SN50", OUT_1 => "01_PushButton"."SE01+NA2006-S1_PB", OUT_2 => "01_PushButton"."SE01+NA2007-S1_PB", OUT_3 => "01_PushButton"."SE01+NA1112-S1_PB", OUT_4 =>, Diag_1 =>, Diag_2 =>, Diag_3 =>, Diag_4 =>, Lamp_1 =>, Lamp_2 =>, Lamp_3 =>, Lamp_4 =>)
   END_RUNG
   // the same network as SCL:
   "n0053-uc12-el001-k30001_SN50_3"(IN_1 := "EMERGENCY PUSH BUTTON PRESSED =SE01+NA2006-S1",   // "00_Push-Button_Input"
                           IN_2 := "EMERGENCY PUSH BUTTON PRESSED =SE01+NA2007-S1",
                           IN_3 := "EMERGENCY PUSH BUTTON PRESSED =SE01+NA1112-S1",
                           ON_Tristate := "06_Settings".Tristate,
                           Bypass_ET200 := "00_Commissioning"."n0053-uc12-el001-k30001_SN50",
                           OUT_1 => "01_PushButton"."SE01+NA2006-S1_PB",
                           OUT_2 => "01_PushButton"."SE01+NA2007-S1_PB",
                           OUT_3 => "01_PushButton"."SE01+NA1112-S1_PB");
END_REGION

REGION Network 48: 50.055 | n0055-uc124-xn10_SN50 [1]
   RUNG wire#powerrail
      "n0055-uc124-xn10_SN50_1"(IN_1 := "EMERGENCY PUSH BUTTON PRESSED =SE01+NA1008-S1", IN_2 := "EMERGENCY PUSH BUTTON PRESSED =SE01+NA1009-S1", IN_3 := "EMERGENCY PUSH BUTTON PRESSED =SE01+NA1010-S1", IN_4 := "EMERGENCY PUSH BUTTON PRESSED =SE01+NA1011-S1", ON_Tristate := "06_Settings".Tristate, ON_Lamp :=, Reset :=, REAC_DELAY :=, Bypass_ET200 := "00_Commissioning"."n0055-uc124-xn10_SN50", OUT_1 => "01_PushButton"."SE01+NA1008-S1_PB", OUT_2 => "01_PushButton"."SE01+NA1009-S1_PB", OUT_3 => "01_PushButton"."SE01+NA1010-S1_PB", OUT_4 => "01_PushButton"."SE01+NA1011-S1_PB", Diag_1 =>, Diag_2 =>, Diag_3 =>, Diag_4 =>, Lamp_1 =>, Lamp_2 =>, Lamp_3 =>, Lamp_4 =>)
   END_RUNG
   // the same network as SCL:
   "n0055-uc124-xn10_SN50_1"(IN_1 := "EMERGENCY PUSH BUTTON PRESSED =SE01+NA1008-S1",   // "00_Push-Button_Input"
                           IN_2 := "EMERGENCY PUSH BUTTON PRESSED =SE01+NA1009-S1",
                           IN_3 := "EMERGENCY PUSH BUTTON PRESSED =SE01+NA1010-S1",
                           IN_4 := "EMERGENCY PUSH BUTTON PRESSED =SE01+NA1011-S1",
                           ON_Tristate := "06_Settings".Tristate,
                           Bypass_ET200 := "00_Commissioning"."n0055-uc124-xn10_SN50",
                           OUT_1 => "01_PushButton"."SE01+NA1008-S1_PB",
                           OUT_2 => "01_PushButton"."SE01+NA1009-S1_PB",
                           OUT_3 => "01_PushButton"."SE01+NA1010-S1_PB",
                           OUT_4 => "01_PushButton"."SE01+NA1011-S1_PB");
END_REGION

REGION Network 49: 50.055 | n0055-uc124-xn10_SN50 [2]
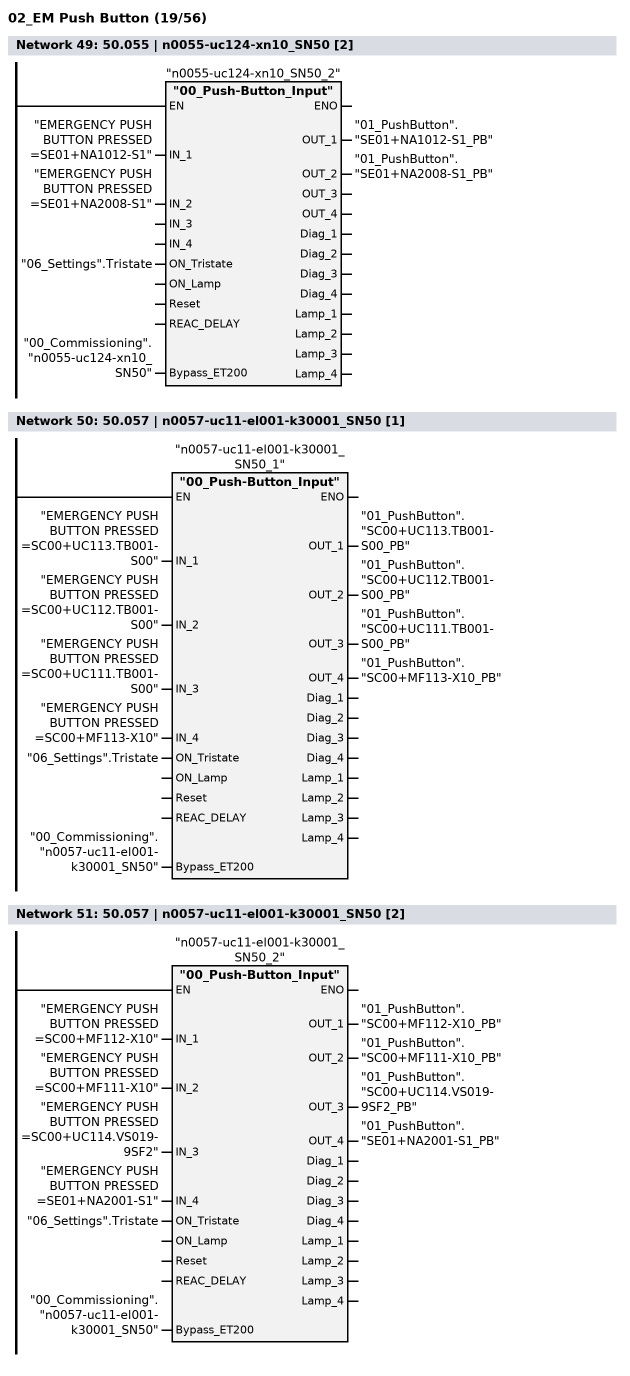
   RUNG wire#powerrail
      "n0055-uc124-xn10_SN50_2"(IN_1 := "EMERGENCY PUSH BUTTON PRESSED =SE01+NA1012-S1", IN_2 := "EMERGENCY PUSH BUTTON PRESSED =SE01+NA2008-S1", IN_3 :=, IN_4 :=, ON_Tristate := "06_Settings".Tristate, ON_Lamp :=, Reset :=, REAC_DELAY :=, Bypass_ET200 := "00_Commissioning"."n0055-uc124-xn10_SN50", OUT_1 => "01_PushButton"."SE01+NA1012-S1_PB", OUT_2 => "01_PushButton"."SE01+NA2008-S1_PB", OUT_3 =>, OUT_4 =>, Diag_1 =>, Diag_2 =>, Diag_3 =>, Diag_4 =>, Lamp_1 =>, Lamp_2 =>, Lamp_3 =>, Lamp_4 =>)
   END_RUNG
   // the same network as SCL:
   "n0055-uc124-xn10_SN50_2"(IN_1 := "EMERGENCY PUSH BUTTON PRESSED =SE01+NA1012-S1",   // "00_Push-Button_Input"
                           IN_2 := "EMERGENCY PUSH BUTTON PRESSED =SE01+NA2008-S1",
                           ON_Tristate := "06_Settings".Tristate,
                           Bypass_ET200 := "00_Commissioning"."n0055-uc124-xn10_SN50",
                           OUT_1 => "01_PushButton"."SE01+NA1012-S1_PB",
                           OUT_2 => "01_PushButton"."SE01+NA2008-S1_PB");
END_REGION

REGION Network 50: 50.057 | n0057-uc11-el001-k30001_SN50 [1]
   RUNG wire#powerrail
      "n0057-uc11-el001-k30001_SN50_1"(IN_1 := "EMERGENCY PUSH BUTTON PRESSED =SC00+UC113.TB001-S00", IN_2 := "EMERGENCY PUSH BUTTON PRESSED =SC00+UC112.TB001-S00", IN_3 := "EMERGENCY PUSH BUTTON PRESSED =SC00+UC111.TB001-S00", IN_4 := "EMERGENCY PUSH BUTTON PRESSED =SC00+MF113-X10", ON_Tristate := "06_Settings".Tristate, ON_Lamp :=, Reset :=, REAC_DELAY :=, Bypass_ET200 := "00_Commissioning"."n0057-uc11-el001-k30001_SN50", OUT_1 => "01_PushButton"."SC00+UC113.TB001-S00_PB", OUT_2 => "01_PushButton"."SC00+UC112.TB001-S00_PB", OUT_3 => "01_PushButton"."SC00+UC111.TB001-S00_PB", OUT_4 => "01_PushButton"."SC00+MF113-X10_PB", Diag_1 =>, Diag_2 =>, Diag_3 =>, Diag_4 =>, Lamp_1 =>, Lamp_2 =>, Lamp_3 =>, Lamp_4 =>)
   END_RUNG
   // the same network as SCL:
   "n0057-uc11-el001-k30001_SN50_1"(IN_1 := "EMERGENCY PUSH BUTTON PRESSED =SC00+UC113.TB001-S00",   // "00_Push-Button_Input"
                           IN_2 := "EMERGENCY PUSH BUTTON PRESSED =SC00+UC112.TB001-S00",
                           IN_3 := "EMERGENCY PUSH BUTTON PRESSED =SC00+UC111.TB001-S00",
                           IN_4 := "EMERGENCY PUSH BUTTON PRESSED =SC00+MF113-X10",
                           ON_Tristate := "06_Settings".Tristate,
                           Bypass_ET200 := "00_Commissioning"."n0057-uc11-el001-k30001_SN50",
                           OUT_1 => "01_PushButton"."SC00+UC113.TB001-S00_PB",
                           OUT_2 => "01_PushButton"."SC00+UC112.TB001-S00_PB",
                           OUT_3 => "01_PushButton"."SC00+UC111.TB001-S00_PB",
                           OUT_4 => "01_PushButton"."SC00+MF113-X10_PB");
END_REGION

REGION Network 51: 50.057 | n0057-uc11-el001-k30001_SN50 [2]
   RUNG wire#powerrail
      "n0057-uc11-el001-k30001_SN50_2"(IN_1 := "EMERGENCY PUSH BUTTON PRESSED =SC00+MF112-X10", IN_2 := "EMERGENCY PUSH BUTTON PRESSED =SC00+MF111-X10", IN_3 := "EMERGENCY PUSH BUTTON PRESSED =SC00+UC114.VS019-9SF2", IN_4 := "EMERGENCY PUSH BUTTON PRESSED =SE01+NA2001-S1", ON_Tristate := "06_Settings".Tristate, ON_Lamp :=, Reset :=, REAC_DELAY :=, Bypass_ET200 := "00_Commissioning"."n0057-uc11-el001-k30001_SN50", OUT_1 => "01_PushButton"."SC00+MF112-X10_PB", OUT_2 => "01_PushButton"."SC00+MF111-X10_PB", OUT_3 => "01_PushButton"."SC00+UC114.VS019-9SF2_PB", OUT_4 => "01_PushButton"."SE01+NA2001-S1_PB", Diag_1 =>, Diag_2 =>, Diag_3 =>, Diag_4 =>, Lamp_1 =>, Lamp_2 =>, Lamp_3 =>, Lamp_4 =>)
   END_RUNG
   // the same network as SCL:
   "n0057-uc11-el001-k30001_SN50_2"(IN_1 := "EMERGENCY PUSH BUTTON PRESSED =SC00+MF112-X10",   // "00_Push-Button_Input"
                           IN_2 := "EMERGENCY PUSH BUTTON PRESSED =SC00+MF111-X10",
                           IN_3 := "EMERGENCY PUSH BUTTON PRESSED =SC00+UC114.VS019-9SF2",
                           IN_4 := "EMERGENCY PUSH BUTTON PRESSED =SE01+NA2001-S1",
                           ON_Tristate := "06_Settings".Tristate,
                           Bypass_ET200 := "00_Commissioning"."n0057-uc11-el001-k30001_SN50",
                           OUT_1 => "01_PushButton"."SC00+MF112-X10_PB",
                           OUT_2 => "01_PushButton"."SC00+MF111-X10_PB",
                           OUT_3 => "01_PushButton"."SC00+UC114.VS019-9SF2_PB",
                           OUT_4 => "01_PushButton"."SE01+NA2001-S1_PB");
END_REGION

REGION Network 52: 50.057 | n0057-uc11-el001-k30001_SN50 [3]
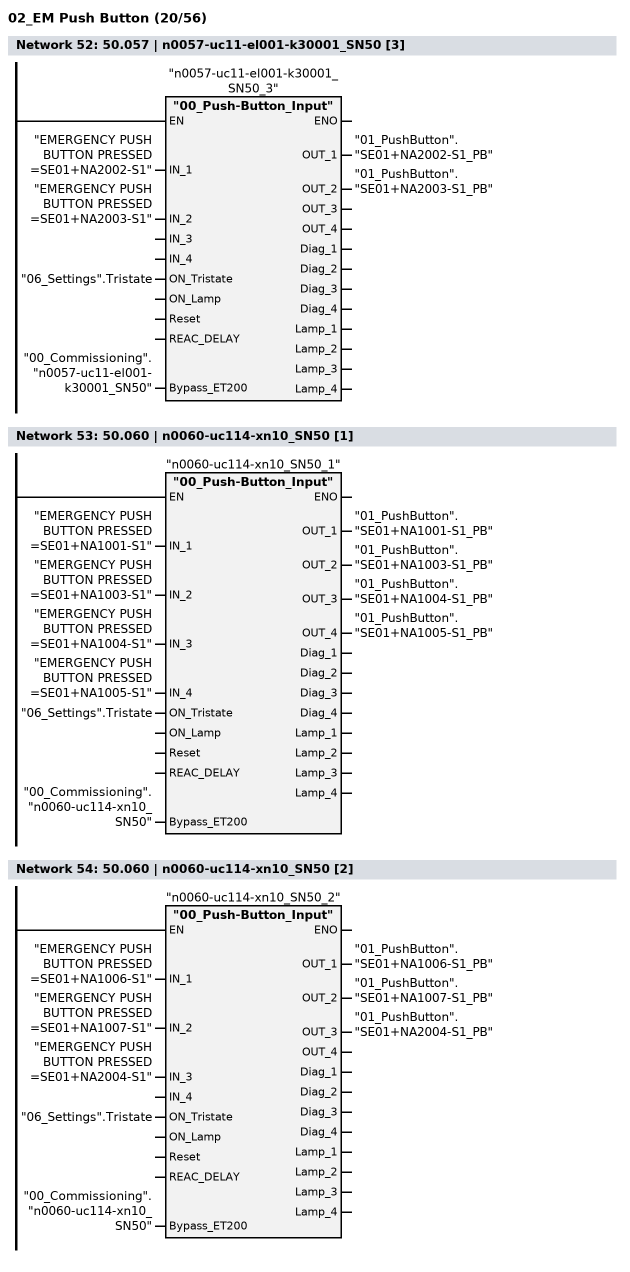
   RUNG wire#powerrail
      "n0057-uc11-el001-k30001_SN50_3"(IN_1 := "EMERGENCY PUSH BUTTON PRESSED =SE01+NA2002-S1", IN_2 := "EMERGENCY PUSH BUTTON PRESSED =SE01+NA2003-S1", IN_3 :=, IN_4 :=, ON_Tristate := "06_Settings".Tristate, ON_Lamp :=, Reset :=, REAC_DELAY :=, Bypass_ET200 := "00_Commissioning"."n0057-uc11-el001-k30001_SN50", OUT_1 => "01_PushButton"."SE01+NA2002-S1_PB", OUT_2 => "01_PushButton"."SE01+NA2003-S1_PB", OUT_3 =>, OUT_4 =>, Diag_1 =>, Diag_2 =>, Diag_3 =>, Diag_4 =>, Lamp_1 =>, Lamp_2 =>, Lamp_3 =>, Lamp_4 =>)
   END_RUNG
   // the same network as SCL:
   "n0057-uc11-el001-k30001_SN50_3"(IN_1 := "EMERGENCY PUSH BUTTON PRESSED =SE01+NA2002-S1",   // "00_Push-Button_Input"
                           IN_2 := "EMERGENCY PUSH BUTTON PRESSED =SE01+NA2003-S1",
                           ON_Tristate := "06_Settings".Tristate,
                           Bypass_ET200 := "00_Commissioning"."n0057-uc11-el001-k30001_SN50",
                           OUT_1 => "01_PushButton"."SE01+NA2002-S1_PB",
                           OUT_2 => "01_PushButton"."SE01+NA2003-S1_PB");
END_REGION

REGION Network 53: 50.060 | n0060-uc114-xn10_SN50 [1]
   RUNG wire#powerrail
      "n0060-uc114-xn10_SN50_1"(IN_1 := "EMERGENCY PUSH BUTTON PRESSED =SE01+NA1001-S1", IN_2 := "EMERGENCY PUSH BUTTON PRESSED =SE01+NA1003-S1", IN_3 := "EMERGENCY PUSH BUTTON PRESSED =SE01+NA1004-S1", IN_4 := "EMERGENCY PUSH BUTTON PRESSED =SE01+NA1005-S1", ON_Tristate := "06_Settings".Tristate, ON_Lamp :=, Reset :=, REAC_DELAY :=, Bypass_ET200 := "00_Commissioning"."n0060-uc114-xn10_SN50", OUT_1 => "01_PushButton"."SE01+NA1001-S1_PB", OUT_2 => "01_PushButton"."SE01+NA1003-S1_PB", OUT_3 => "01_PushButton"."SE01+NA1004-S1_PB", OUT_4 => "01_PushButton"."SE01+NA1005-S1_PB", Diag_1 =>, Diag_2 =>, Diag_3 =>, Diag_4 =>, Lamp_1 =>, Lamp_2 =>, Lamp_3 =>, Lamp_4 =>)
   END_RUNG
   // the same network as SCL:
   "n0060-uc114-xn10_SN50_1"(IN_1 := "EMERGENCY PUSH BUTTON PRESSED =SE01+NA1001-S1",   // "00_Push-Button_Input"
                           IN_2 := "EMERGENCY PUSH BUTTON PRESSED =SE01+NA1003-S1",
                           IN_3 := "EMERGENCY PUSH BUTTON PRESSED =SE01+NA1004-S1",
                           IN_4 := "EMERGENCY PUSH BUTTON PRESSED =SE01+NA1005-S1",
                           ON_Tristate := "06_Settings".Tristate,
                           Bypass_ET200 := "00_Commissioning"."n0060-uc114-xn10_SN50",
                           OUT_1 => "01_PushButton"."SE01+NA1001-S1_PB",
                           OUT_2 => "01_PushButton"."SE01+NA1003-S1_PB",
                           OUT_3 => "01_PushButton"."SE01+NA1004-S1_PB",
                           OUT_4 => "01_PushButton"."SE01+NA1005-S1_PB");
END_REGION

REGION Network 54: 50.060 | n0060-uc114-xn10_SN50 [2]
   RUNG wire#powerrail
      "n0060-uc114-xn10_SN50_2"(IN_1 := "EMERGENCY PUSH BUTTON PRESSED =SE01+NA1006-S1", IN_2 := "EMERGENCY PUSH BUTTON PRESSED =SE01+NA1007-S1", IN_3 := "EMERGENCY PUSH BUTTON PRESSED =SE01+NA2004-S1", IN_4 :=, ON_Tristate := "06_Settings".Tristate, ON_Lamp :=, Reset :=, REAC_DELAY :=, Bypass_ET200 := "00_Commissioning"."n0060-uc114-xn10_SN50", OUT_1 => "01_PushButton"."SE01+NA1006-S1_PB", OUT_2 => "01_PushButton"."SE01+NA1007-S1_PB", OUT_3 => "01_PushButton"."SE01+NA2004-S1_PB", OUT_4 =>, Diag_1 =>, Diag_2 =>, Diag_3 =>, Diag_4 =>, Lamp_1 =>, Lamp_2 =>, Lamp_3 =>, Lamp_4 =>)
   END_RUNG
   // the same network as SCL:
   "n0060-uc114-xn10_SN50_2"(IN_1 := "EMERGENCY PUSH BUTTON PRESSED =SE01+NA1006-S1",   // "00_Push-Button_Input"
                           IN_2 := "EMERGENCY PUSH BUTTON PRESSED =SE01+NA1007-S1",
                           IN_3 := "EMERGENCY PUSH BUTTON PRESSED =SE01+NA2004-S1",
                           ON_Tristate := "06_Settings".Tristate,
                           Bypass_ET200 := "00_Commissioning"."n0060-uc114-xn10_SN50",
                           OUT_1 => "01_PushButton"."SE01+NA1006-S1_PB",
                           OUT_2 => "01_PushButton"."SE01+NA1007-S1_PB",
                           OUT_3 => "01_PushButton"."SE01+NA2004-S1_PB");
END_REGION

REGION Network 55: 50.028 | n0028-uc17-el001-k30001_SN50 [1]
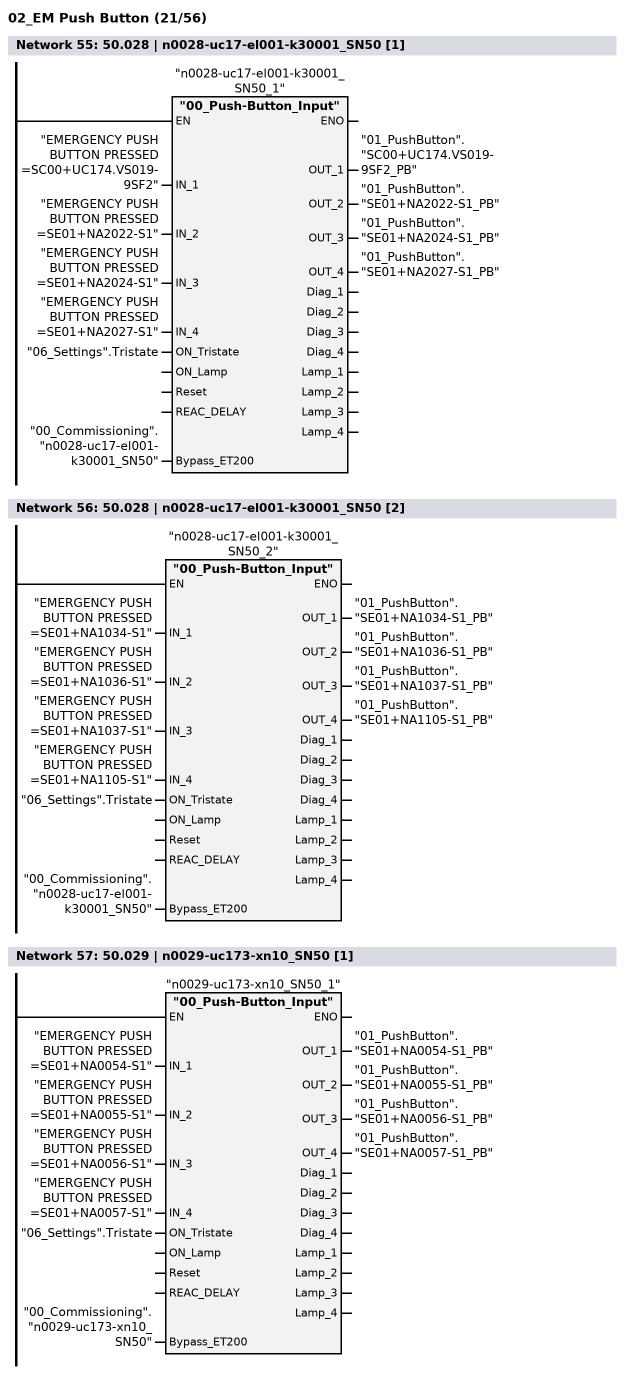
   RUNG wire#powerrail
      "n0028-uc17-el001-k30001_SN50_1"(IN_1 := "EMERGENCY PUSH BUTTON PRESSED =SC00+UC174.VS019-9SF2", IN_2 := "EMERGENCY PUSH BUTTON PRESSED =SE01+NA2022-S1", IN_3 := "EMERGENCY PUSH BUTTON PRESSED =SE01+NA2024-S1", IN_4 := "EMERGENCY PUSH BUTTON PRESSED =SE01+NA2027-S1", ON_Tristate := "06_Settings".Tristate, ON_Lamp :=, Reset :=, REAC_DELAY :=, Bypass_ET200 := "00_Commissioning"."n0028-uc17-el001-k30001_SN50", OUT_1 => "01_PushButton"."SC00+UC174.VS019-9SF2_PB", OUT_2 => "01_PushButton"."SE01+NA2022-S1_PB", OUT_3 => "01_PushButton"."SE01+NA2024-S1_PB", OUT_4 => "01_PushButton"."SE01+NA2027-S1_PB", Diag_1 =>, Diag_2 =>, Diag_3 =>, Diag_4 =>, Lamp_1 =>, Lamp_2 =>, Lamp_3 =>, Lamp_4 =>)
   END_RUNG
   // the same network as SCL:
   "n0028-uc17-el001-k30001_SN50_1"(IN_1 := "EMERGENCY PUSH BUTTON PRESSED =SC00+UC174.VS019-9SF2",   // "00_Push-Button_Input"
                           IN_2 := "EMERGENCY PUSH BUTTON PRESSED =SE01+NA2022-S1",
                           IN_3 := "EMERGENCY PUSH BUTTON PRESSED =SE01+NA2024-S1",
                           IN_4 := "EMERGENCY PUSH BUTTON PRESSED =SE01+NA2027-S1",
                           ON_Tristate := "06_Settings".Tristate,
                           Bypass_ET200 := "00_Commissioning"."n0028-uc17-el001-k30001_SN50",
                           OUT_1 => "01_PushButton"."SC00+UC174.VS019-9SF2_PB",
                           OUT_2 => "01_PushButton"."SE01+NA2022-S1_PB",
                           OUT_3 => "01_PushButton"."SE01+NA2024-S1_PB",
                           OUT_4 => "01_PushButton"."SE01+NA2027-S1_PB");
END_REGION

REGION Network 56: 50.028 | n0028-uc17-el001-k30001_SN50 [2]
   RUNG wire#powerrail
      "n0028-uc17-el001-k30001_SN50_2"(IN_1 := "EMERGENCY PUSH BUTTON PRESSED =SE01+NA1034-S1", IN_2 := "EMERGENCY PUSH BUTTON PRESSED =SE01+NA1036-S1", IN_3 := "EMERGENCY PUSH BUTTON PRESSED =SE01+NA1037-S1", IN_4 := "EMERGENCY PUSH BUTTON PRESSED =SE01+NA1105-S1", ON_Tristate := "06_Settings".Tristate, ON_Lamp :=, Reset :=, REAC_DELAY :=, Bypass_ET200 := "00_Commissioning"."n0028-uc17-el001-k30001_SN50", OUT_1 => "01_PushButton"."SE01+NA1034-S1_PB", OUT_2 => "01_PushButton"."SE01+NA1036-S1_PB", OUT_3 => "01_PushButton"."SE01+NA1037-S1_PB", OUT_4 => "01_PushButton"."SE01+NA1105-S1_PB", Diag_1 =>, Diag_2 =>, Diag_3 =>, Diag_4 =>, Lamp_1 =>, Lamp_2 =>, Lamp_3 =>, Lamp_4 =>)
   END_RUNG
   // the same network as SCL:
   "n0028-uc17-el001-k30001_SN50_2"(IN_1 := "EMERGENCY PUSH BUTTON PRESSED =SE01+NA1034-S1",   // "00_Push-Button_Input"
                           IN_2 := "EMERGENCY PUSH BUTTON PRESSED =SE01+NA1036-S1",
                           IN_3 := "EMERGENCY PUSH BUTTON PRESSED =SE01+NA1037-S1",
                           IN_4 := "EMERGENCY PUSH BUTTON PRESSED =SE01+NA1105-S1",
                           ON_Tristate := "06_Settings".Tristate,
                           Bypass_ET200 := "00_Commissioning"."n0028-uc17-el001-k30001_SN50",
                           OUT_1 => "01_PushButton"."SE01+NA1034-S1_PB",
                           OUT_2 => "01_PushButton"."SE01+NA1036-S1_PB",
                           OUT_3 => "01_PushButton"."SE01+NA1037-S1_PB",
                           OUT_4 => "01_PushButton"."SE01+NA1105-S1_PB");
END_REGION

REGION Network 57: 50.029 | n0029-uc173-xn10_SN50 [1]
   RUNG wire#powerrail
      "n0029-uc173-xn10_SN50_1"(IN_1 := "EMERGENCY PUSH BUTTON PRESSED =SE01+NA0054-S1", IN_2 := "EMERGENCY PUSH BUTTON PRESSED =SE01+NA0055-S1", IN_3 := "EMERGENCY PUSH BUTTON PRESSED =SE01+NA0056-S1", IN_4 := "EMERGENCY PUSH BUTTON PRESSED =SE01+NA0057-S1", ON_Tristate := "06_Settings".Tristate, ON_Lamp :=, Reset :=, REAC_DELAY :=, Bypass_ET200 := "00_Commissioning"."n0029-uc173-xn10_SN50", OUT_1 => "01_PushButton"."SE01+NA0054-S1_PB", OUT_2 => "01_PushButton"."SE01+NA0055-S1_PB", OUT_3 => "01_PushButton"."SE01+NA0056-S1_PB", OUT_4 => "01_PushButton"."SE01+NA0057-S1_PB", Diag_1 =>, Diag_2 =>, Diag_3 =>, Diag_4 =>, Lamp_1 =>, Lamp_2 =>, Lamp_3 =>, Lamp_4 =>)
   END_RUNG
   // the same network as SCL:
   "n0029-uc173-xn10_SN50_1"(IN_1 := "EMERGENCY PUSH BUTTON PRESSED =SE01+NA0054-S1",   // "00_Push-Button_Input"
                           IN_2 := "EMERGENCY PUSH BUTTON PRESSED =SE01+NA0055-S1",
                           IN_3 := "EMERGENCY PUSH BUTTON PRESSED =SE01+NA0056-S1",
                           IN_4 := "EMERGENCY PUSH BUTTON PRESSED =SE01+NA0057-S1",
                           ON_Tristate := "06_Settings".Tristate,
                           Bypass_ET200 := "00_Commissioning"."n0029-uc173-xn10_SN50",
                           OUT_1 => "01_PushButton"."SE01+NA0054-S1_PB",
                           OUT_2 => "01_PushButton"."SE01+NA0055-S1_PB",
                           OUT_3 => "01_PushButton"."SE01+NA0056-S1_PB",
                           OUT_4 => "01_PushButton"."SE01+NA0057-S1_PB");
END_REGION

REGION Network 58: 50.029 | n0029-uc173-xn10_SN50 [2]
